ACTION IOFilter_Action:
;
(* Update Functions for pin 1.9 *)

    (* AI filtering for pin X1.09 *)
        AI_u16_DrivetrainTemp_AI := AI_MeanValue(AI_ARR_INDEX,ADR(AI_ARR_u16_DrivetrainTemp_AI),1,50,10);
        AIPU_u16_DrivetrainTemp_AI := AI_MeanValue(AI_ARR_INDEX,ADR(AIPU_ARR_u16_DrivetrainTemp_AI),1,50,10);


(* Update Functions for pin 1.10 *)

    (* AI filtering for pin X1.10 *)
        AI_u16_ChargePlugPresent_AI := AI_MeanValue(AI_ARR_INDEX,ADR(AI_ARR_u16_ChargePlugPresent_AI),1,50,10);
        AIPU_u16_ChargePlugPresent_AI := AI_MeanValue(AI_ARR_INDEX,ADR(AIPU_ARR_u16_ChargePlugPresent_AI),1,50,10);


(* Update Functions for pin 1.11 *)

     (* Debounce filtering to raw DI value of pin 1.11 *)
     G_DebounceDI_q_BatteryInterlockIn_DI(i_In:=DI_RAW_q_BatteryInterlockIn_DI,i_Delay:=30);
     DI_q_BatteryInterlockIn_DI:=G_DebounceDI_q_BatteryInterlockIn_DI.o_Out;

(* Update Functions for pin 1.12 *)

(* Update Functions for pin 1.20 *)

    (* AI filtering for pin X1.20 *)
        AI_u16_Heater1Temperature_AI := AI_MeanValue(AI_ARR_INDEX,ADR(AI_ARR_u16_Heater1Temperature_AI),1,50,10);
        AIPU_u16_Heater1Temperature_AI := AI_MeanValue(AI_ARR_INDEX,ADR(AIPU_ARR_u16_Heater1Temperature_AI),1,50,10);


(* Update Functions for pin 1.21 *)

    (* AI filtering for pin X1.21 *)
        AI_u16_Heater2Temperature_AI := AI_MeanValue(AI_ARR_INDEX,ADR(AI_ARR_u16_Heater2Temperature_AI),1,50,10);
        AIPU_u16_Heater2Temperature_AI := AI_MeanValue(AI_ARR_INDEX,ADR(AIPU_ARR_u16_Heater2Temperature_AI),1,50,10);


(* Update Functions for pin 1.22 *)

(* Update Functions for pin 1.23 *)

(* Update Functions for pin 1.29 *)

(* Update Functions for pin 1.30 *)

(* Update Functions for pin 1.31 *)

(* Update Functions for pin 1.32 *)

(* Update Functions for pin 1.33 *)

(* Update Functions for pin 1.34 *)

(* Update Functions for pin 1.35 *)

(* Update Functions for pin 2.6 *)

     (* Debounce filtering to raw DI value of pin 2.6 *)
     G_DebounceDI_q_Battery1ChargeRq_DI(i_In:=DI_RAW_q_Battery1ChargeRq_DI,i_Delay:=30);
     DI_q_Battery1ChargeRq_DI:=G_DebounceDI_q_Battery1ChargeRq_DI.o_Out;

(* Update Functions for pin 2.7 *)

     (* Debounce filtering to raw DI value of pin 2.7 *)
     G_DebounceDI_q_Battery1DiscahrgeRq_DI(i_In:=DI_RAW_q_Battery1DiscahrgeRq_DI,i_Delay:=30);
     DI_q_Battery1DiscahrgeRq_DI:=G_DebounceDI_q_Battery1DiscahrgeRq_DI.o_Out;

(* Update Functions for pin 2.8 *)

     (* Debounce filtering to raw DI value of pin 2.8 *)
     G_DebounceDI_q_Battery2ChargeRq_DI(i_In:=DI_RAW_q_Battery2ChargeRq_DI,i_Delay:=30);
     DI_q_Battery2ChargeRq_DI:=G_DebounceDI_q_Battery2ChargeRq_DI.o_Out;

(* Update Functions for pin 2.9 *)

     (* Debounce filtering to raw DI value of pin 2.9 *)
     G_DebounceDI_q_Batter2DischargeRq_DI(i_In:=DI_RAW_q_Batter2DischargeRq_DI,i_Delay:=30);
     DI_q_Batter2DischargeRq_DI:=G_DebounceDI_q_Batter2DischargeRq_DI.o_Out;

(* Update Functions for pin 2.13 *)

(* Update Functions for pin 2.14 *)

(* Update Functions for pin 2.15 *)

(* Update Functions for pin 2.17 *)

     (* Debounce filtering to raw DI value of pin 2.17 *)
     G_DebounceDI_q_ChargePlugLockStatus_DI(i_In:=DI_RAW_q_ChargePlugLockStatus_DI,i_Delay:=30);
     DI_q_ChargePlugLockStatus_DI:=G_DebounceDI_q_ChargePlugLockStatus_DI.o_Out;

(* Update Functions for pin 2.17 *)

(* Update Functions for pin 2.18 *)

(* Update Functions for pin 2.19 *)

(* Update Functions for pin 2.20 *)

(* Update Functions for pin 2.23 *)

    (* AI filtering for pin X2.23 *)
        AI_u16_HeaterDiagnose_AI := AI_MeanValue(AI_ARR_INDEX,ADR(AI_ARR_u16_HeaterDiagnose_AI),1,50,10);
        AIPU_u16_HeaterDiagnose_AI := AI_MeanValue(AI_ARR_INDEX,ADR(AIPU_ARR_u16_HeaterDiagnose_AI),1,50,10);


(* Update Functions for pin 2.26 *)

(* Update Functions for pin 2.27 *)

(* Update Functions for pin 2.28 *)

(* Update Functions for pin 2.29 *)

(* Update Functions for pin 2.30 *)

(* Update Functions for pin 2.31 *)

(* Update Functions for pin 2.32 *)

(* Update Functions for pin 2.33 *)

(* Update Functions for pin 2.34 *)

(* Update Functions for pin 2.35 *)

(* Update Functions for pin 3.5 *)

     (* Debounce filtering to raw DI value of pin 3.5 *)
     G_DebounceDI_q_DirectionSwitch_ReverseCrawl_DI(i_In:=DI_RAW_q_DirectionSwitch_ReverseCrawl_DI,i_Delay:=30);
     DI_q_DirectionSwitch_ReverseCrawl_DI:=G_DebounceDI_q_DirectionSwitch_ReverseCrawl_DI.o_Out;

(* Update Functions for pin 3.6 *)

     (* Debounce filtering to raw DI value of pin 3.6 *)
     G_DebounceDI_q_DirectionSwitch_Drive_DI(i_In:=DI_RAW_q_DirectionSwitch_Drive_DI,i_Delay:=30);
     DI_q_DirectionSwitch_Drive_DI:=G_DebounceDI_q_DirectionSwitch_Drive_DI.o_Out;

(* Update Functions for pin 3.7 *)

     (* Debounce filtering to raw DI value of pin 3.7 *)
     G_DebounceDI_q_IlluminiationStatsus_DI(i_In:=DI_RAW_q_IlluminiationStatsus_DI,i_Delay:=30);
     DI_q_IlluminiationStatsus_DI:=G_DebounceDI_q_IlluminiationStatsus_DI.o_Out;

(* Update Functions for pin 3.8 *)

     (* Debounce filtering to raw DI value of pin 3.8 *)
     G_DebounceDI_q_DirectionSwitch_Reverse_DI(i_In:=DI_RAW_q_DirectionSwitch_Reverse_DI,i_Delay:=30);
     DI_q_DirectionSwitch_Reverse_DI:=G_DebounceDI_q_DirectionSwitch_Reverse_DI.o_Out;

(* Update Functions for pin 3.9 *)

     (* Debounce filtering to raw DI value of pin 3.9 *)
     G_DebounceDI_q_DirectionSwitch_DriveCrawl_DI(i_In:=DI_RAW_q_DirectionSwitch_DriveCrawl_DI,i_Delay:=30);
     DI_q_DirectionSwitch_DriveCrawl_DI:=G_DebounceDI_q_DirectionSwitch_DriveCrawl_DI.o_Out;

(* Update Functions for pin 3.10 *)

(* Update Functions for pin 3.11 *)

     (* Debounce filtering to raw DI value of pin 3.11 *)
     G_DebounceDI_q_DirectionSwitch_Neutral_DI(i_In:=DI_RAW_q_DirectionSwitch_Neutral_DI,i_Delay:=30);
     DI_q_DirectionSwitch_Neutral_DI:=G_DebounceDI_q_DirectionSwitch_Neutral_DI.o_Out;

(* Update Functions for pin 3.12 *)

     (* Debounce filtering to raw DI value of pin 3.12 *)
     G_DebounceDI_q_DoorOpen_DI(i_In:=DI_RAW_q_DoorOpen_DI,i_Delay:=30);
     DI_q_DoorOpen_DI:=G_DebounceDI_q_DoorOpen_DI.o_Out;

(* Update Functions for pin 3.14 *)

    (* AI filtering for pin X3.14 *)
        AI_u16_HeaterDiagnose2_AI := AI_MeanValue(AI_ARR_INDEX,ADR(AI_ARR_u16_HeaterDiagnose2_AI),1,50,10);
        AIPU_u16_HeaterDiagnose2_AI := AI_MeanValue(AI_ARR_INDEX,ADR(AIPU_ARR_u16_HeaterDiagnose2_AI),1,50,10);


(* Update Functions for pin 3.15 *)

    (* AI filtering for pin X3.15 *)
        AI_u16_VehicleThrottlePedal1_AI := AI_MeanValue(AI_ARR_INDEX,ADR(AI_ARR_u16_VehicleThrottlePedal1_AI),1,50,10);
        AIPU_u16_VehicleThrottlePedal1_AI := AI_MeanValue(AI_ARR_INDEX,ADR(AIPU_ARR_u16_VehicleThrottlePedal1_AI),1,50,10);



(* Update Functions for pin 3.16 *)

    (* AI filtering for pin X3.16 *)
        AI_u16_VehicleThrottlePedal2_AI := AI_MeanValue(AI_ARR_INDEX,ADR(AI_ARR_u16_VehicleThrottlePedal2_AI),1,50,10);
        AIPU_u16_VehicleThrottlePedal2_AI := AI_MeanValue(AI_ARR_INDEX,ADR(AIPU_ARR_u16_VehicleThrottlePedal2_AI),1,50,10);



(* Update Functions for pin 3.17 *)

(* Update Functions for pin 3.18 *)

(* Update Functions for pin 3.19 *)

(* Update Functions for pin 3.21 *)

(* Update Functions for pin 3.22 *)

     (* Debounce filtering to raw DI value of pin 3.22 *)
     G_DebounceDI_q_VehicleKL15_DI(i_In:=DI_RAW_q_VehicleKL15_DI,i_Delay:=30);
     DI_q_VehicleKL15_DI:=G_DebounceDI_q_VehicleKL15_DI.o_Out;

(* Update Functions for pin 3.23 *)

     (* Debounce filtering to raw DI value of pin 3.23 *)
     G_DebounceDI_q_VehicleKL51_DI(i_In:=DI_RAW_q_VehicleKL51_DI,i_Delay:=30);
     DI_q_VehicleKL51_DI:=G_DebounceDI_q_VehicleKL51_DI.o_Out;

(* Update Functions for pin 3.26 *)

(* Update Functions for pin 3.27 *)

(* Update Functions for pin 3.28 *)

    (* Debounce filtering to raw DI value of pin 3.28 *)
        G_DebounceDI_q_HeaterIn_DI(i_In:=DI_RAW_q_HeaterIn_DI,i_Delay:=30);
        DI_q_HeaterIn_DI:=G_DebounceDI_q_HeaterIn_DI.o_Out;

(* Update Functions for pin 3.29 *)

    (* AI filtering for output voltage measurement in pin X3.29 *)
        AI_q_HeaterOut_DI_Ai := AI_MeanValue(AI_ARR_INDEX,ADR(AI_ARR_q_HeaterOut_DI),1,50,10);


(* Update Functions for pin 3.30 *)

    (* AI filtering for output voltage measurement in pin X3.30 *)
        AI_q_DrivetrainInverterRf1_DO_Ai := AI_MeanValue(AI_ARR_INDEX,ADR(AI_ARR_q_DrivetrainInverterRf1_DO),1,50,10);

(* Update Functions for pin 3.31 *)

    (* AI filtering for output voltage measurement in pin X3.31 *)
        AI_q_DrivetrainInverterRf2_DO_Ai := AI_MeanValue(AI_ARR_INDEX,ADR(AI_ARR_q_DrivetrainInverterRf2_DO),1,50,10);

(* Update Functions for pin 3.32 *)

    (* AI filtering for output voltage measurement in pin X3.32 *)
        AI_q_DrivetrainDCDCInhibit_DO_Ai := AI_MeanValue(AI_ARR_INDEX,ADR(AI_ARR_q_DrivetrainDCDCInhibit_DO),1,50,10);


(* Update Functions for pin 3.33 *)

    (* AI filtering for output voltage measurement in pin X3.33 *)
        AI_q_ChargePlugLED_Green_DO_Ai := AI_MeanValue(AI_ARR_INDEX,ADR(AI_ARR_q_ChargePlugLED_Green_DO),1,50,10);

(* Update Functions for pin 3.34 *)

    (* AI filtering for output voltage measurement in pin X3.34 *)
        AI_q_ChargePlugLED_Blue_DO_Ai := AI_MeanValue(AI_ARR_INDEX,ADR(AI_ARR_q_ChargePlugLED_Blue_DO),1,50,10);

(* Update Functions for pin 3.35 *)

    (* AI filtering for output voltage measurement in pin X3.35 *)
        AI_q_ChargePlugLED_Red_DO_Ai := AI_MeanValue(AI_ARR_INDEX,ADR(AI_ARR_q_ChargePlugLED_Red_DO),1,50,10);
END_ACTION

ACTION IOHandleOutputs_Action:
;

(* AI over current protection for pin X1.09 *)
   IF AI_SET_mA_u16_DrivetrainTemp_AI = TRUE THEN
        (* mA resistor connected set mode correctly *)
        G_AIprotection_X1_09(i_AiInmAMode:= TRUE);
   END_IF
   G_AIprotection_X1_09(
                                                      i_PullUpVoltage := AIPU_RAW_u16_DrivetrainTemp_AI,
                                                      o_ModeSelection =>AI_SET_mA_u16_DrivetrainTemp_AI,
                                                      o_OverCurrentError =>ERR_FLAG_IO_AI_OVER_CURRENT_X1_09);

(* AI over current protection for pin X1.10 *)
   IF AI_SET_mA_u16_ChargePlugPresent_AI = TRUE THEN
        (* mA resistor connected set mode correctly *)
        G_AIprotection_X1_10(i_AiInmAMode:= TRUE);
   END_IF
   G_AIprotection_X1_10(
                                                      i_PullUpVoltage := AIPU_RAW_u16_ChargePlugPresent_AI,
                                                      o_ModeSelection =>AI_SET_mA_u16_ChargePlugPresent_AI,
                                                      o_OverCurrentError =>ERR_FLAG_IO_AI_OVER_CURRENT_X1_10);

(* AI over current protection for pin X1.20 *)
   IF AI_SET_mA_u16_Heater1Temperature_AI = TRUE THEN
        (* mA resistor connected set mode correctly *)
        G_AIprotection_X1_20(i_AiInmAMode:= TRUE);
   END_IF
   G_AIprotection_X1_20(
                                                      i_PullUpVoltage := AIPU_RAW_u16_Heater1Temperature_AI,
                                                      o_ModeSelection =>AI_SET_mA_u16_Heater1Temperature_AI,
                                                      o_OverCurrentError =>ERR_FLAG_IO_AI_OVER_CURRENT_X1_20);

(* AI over current protection for pin X1.20 *)
   IF AI_SET_mA_u16_Heater2Temperature_AI = TRUE THEN
        (* mA resistor connected set mode correctly *)
        G_AIprotection_X1_21(i_AiInmAMode:= TRUE);
   END_IF
   G_AIprotection_X1_21(
                                                      i_PullUpVoltage := AIPU_RAW_u16_Heater2Temperature_AI,
                                                      o_ModeSelection =>AI_SET_mA_u16_Heater2Temperature_AI,
                                                      o_OverCurrentError =>ERR_FLAG_IO_AI_OVER_CURRENT_X1_21);

(* AI over current protection for pin X2.23 *)
   IF AI_SET_mA_u16_HeaterDiagnose_AI = TRUE THEN
        (* mA resistor connected set mode correctly *)
        G_AIprotection_X2_23(i_AiInmAMode:= TRUE);
   END_IF
   G_AIprotection_X2_23(
                                                      i_PullUpVoltage := AIPU_RAW_u16_HeaterDiagnose_AI,
                                                      o_ModeSelection =>AI_SET_mA_u16_HeaterDiagnose_AI,
                                                      o_OverCurrentError =>ERR_FLAG_IO_AI_OVER_CURRENT_X2_23);

(* AI over current protection for pin X3.14 *)
   IF AI_SET_mA_u16_HeaterDiagnose2_AI = TRUE THEN
        (* mA resistor connected set mode correctly *)
        G_AIprotection_X3_14(i_AiInmAMode:= TRUE);
   END_IF
   G_AIprotection_X3_14(
                                                      i_PullUpVoltage := AIPU_RAW_u16_HeaterDiagnose2_AI,
                                                      o_ModeSelection =>AI_SET_mA_u16_HeaterDiagnose2_AI,
                                                      o_OverCurrentError =>ERR_FLAG_IO_AI_OVER_CURRENT_X3_14);

(* AI over current protection for pin X3.15 *)
   IF AI_SET_mA_u16_VehicleThrottlePedal1_AI = TRUE THEN
        (* mA resistor connected set mode correctly *)
        G_AIprotection_X3_15(i_AiInmAMode:= TRUE);
   END_IF
   G_AIprotection_X3_15(
                                                      i_PullUpVoltage := AIPU_RAW_u16_VehicleThrottlePedal1_AI,
                                                      o_ModeSelection =>AI_SET_mA_u16_VehicleThrottlePedal1_AI,
                                                      o_OverCurrentError =>ERR_FLAG_IO_AI_OVER_CURRENT_X3_15);

(* AI over current protection for pin X3.16 *)
   IF AI_SET_mA_u16_VehicleThrottlePedal2_AI = TRUE THEN
        (* mA resistor connected set mode correctly *)
        G_AIprotection_X3_16(i_AiInmAMode:= TRUE);
   END_IF
   G_AIprotection_X3_16(
                                                      i_PullUpVoltage := AIPU_RAW_u16_VehicleThrottlePedal2_AI,
                                                      o_ModeSelection =>AI_SET_mA_u16_VehicleThrottlePedal2_AI,
                                                      o_OverCurrentError =>ERR_FLAG_IO_AI_OVER_CURRENT_X3_16);
END_ACTION

ACTION Main_Application_Action:
(* Call user application *)
Main();
END_ACTION

ACTION Other_Action:
// Target specific. Not available.
END_ACTION

ACTION Other_EpecOut_Action:
(* tag EPEC_OUT_OTHER *)

(* If reset flag set --> restart unit *)
IF G_RESET_MODULE THEN
    EPEC_5000EXT.BOOT_APPLICATION_KILL_RTS();
END_IF

(* Block actions if voltage level is under defined limit *)
IF G_HWDiagnostics.o_SupplyVoltage1 > G_LowLimitForParameterSaving THEN

	
    IF G_CounterRestoreCmdOld<> G_SaveOD_RestoreCommsCounter THEN 
         (* Restore command given trough CANopen *)
         G_CounterRestoreCmdOld := G_SaveOD_RestoreCommsCounter;   
         SystemParameters.RestoreDefaultData();
         G_SystemInfo.EthernetConfiguration := SystemParameters.i_Ethernet;  
         G_SystemInfo.CAN1_Comms := SystemParameters.i_CAN1;
         G_SystemInfo.CAN2_Comms := SystemParameters.i_CAN2;      
         G_SystemInfo.CAN3_Comms := SystemParameters.i_CAN3;      
         G_SystemInfo.CAN4_Comms := SystemParameters.i_CAN4;      
    END_IF
    
    IF G_CounterSaveCmdOld  <> G_SaveOD_SaveCommsCounter THEN
        (* Save command given trough CANopen *)
        G_CounterSaveCmdOld  := G_SaveOD_SaveCommsCounter;
        SystemParameters.i_Ethernet := G_SystemInfo.EthernetConfiguration;
        SystemParameters.i_CAN1 := G_SystemInfo.CAN1_Comms;
        SystemParameters.i_CAN2 := G_SystemInfo.CAN2_Comms;
        SystemParameters.i_CAN3 := G_SystemInfo.CAN3_Comms;
        SystemParameters.i_CAN4 := G_SystemInfo.CAN4_Comms;
        SystemParameters.WriteData();
    END_IF
END_IF
END_ACTION

END_PROGRAM

// Application/UserCode/Functions/Update
(*==============================================================================================================*)
(*     Function to handle state updates                                                                         *)
(*==============================================================================================================*)
FUNCTION Update : BOOL
VAR_INPUT
 ptUp        : POINTER TO tUpdate; // Pointer to screen update

END_VAR
VAR
END_VAR

(*==============================================================================================================*)
(*     Function to handle state updates                                                                         *)
(*==============================================================================================================*)
IF (ptUp^.Next <> ptUp^.Step) THEN                         // New State Requested?	
	ptUp^.Last			:= ptUp^.Step;                     // Save Current State
	ptUp^.Step			:= ptUp^.Next;                     // Set New State
	ptUp^.Seq  			:= (ptUp^.Seq * 256) + ptUp^.Next; // Shift In New State
	ptUp^.Tmr			:= 0;                              // Reset State Timer
ELSIF (ptUp^.Tmr <> 65535) THEN                            // Timer Less than max?
	ptUp^.Tmr			:= (ptUp^.Tmr + 1);                // Increment Timer
END_IF

END_FUNCTION

// Application/UserCode/Main Program/MainInit
PROGRAM MainInit
VAR_OUTPUT
	o_MainInitReady: BOOL := FALSE;
END_VAR


(*Check if CAN bitrate in device communication parameters is 500kbit/s.
If not, set it to 500 kbit/s *)
EPEC_5050INT.SystemParameters.ReadData();
IF EPEC_5050INT.SystemParameters.i_CAN1[3] <> gu16_CAN1_BaudRate THEN
                             EPEC_5050INT.SystemParameters.i_CAN1[3] := gu16_CAN1_BaudRate;
                             EPEC_5050INT.SystemParameters.WriteData();
END_IF
IF EPEC_5050INT.SystemParameters.i_CAN2[3] <> gu16_CAN2_BaudRate THEN
                             EPEC_5050INT.SystemParameters.i_CAN2[3] := gu16_CAN2_BaudRate;
                             EPEC_5050INT.SystemParameters.WriteData();
END_IF
IF EPEC_5050INT.SystemParameters.i_CAN3[3] <> gu16_CAN3_BaudRate THEN
                             EPEC_5050INT.SystemParameters.i_CAN3[3] := gu16_CAN3_BaudRate;
                             EPEC_5050INT.SystemParameters.WriteData();
END_IF
IF EPEC_5050INT.SystemParameters.i_CAN4[3] <> gu16_CAN4_BaudRate THEN
                             EPEC_5050INT.SystemParameters.i_CAN4[3] := gu16_CAN4_BaudRate;
                             EPEC_5050INT.SystemParameters.WriteData();
END_IF

o_MainInitReady := TRUE;

END_PROGRAM

// Application/UserCode/Main Program/Main
PROGRAM Main
VAR
	hq_ManualChangeBaud	:	BOOL;
	hton_Timer	:	TON;
END_VAR

/// User code should be added to POU named as Main.
(*Reallocation of Outputs to correct variables*)
IO_Reconfiguration();


(*Check to make sure that the component selection hasn't been changed*)
ComponentSelection();

(*******************************************************)
(*Receive Routines*)
Sevcon_Steer_Rx();
Sevcon2_Rx();
Brusa1_Rx();
Brusa2_Rx();
MCU_Rx();
OrionBMS1_Rx();
OrionBMS2_Rx();
BELDCDC_Rx();
BELDCDC_Tx();
BELDCDC_TxConversion();
HMI_Rx();
CAN1_Rx();
CAN3_Rx();
CAN4_Rx();
ePTO_Rx();
Chassis_Parameters();
Cooling_Fan();
(*******************************************************)
(*Control*)
FaultDetection();
System_StateSpace();
ContactorControl();
GearSelection();
Dennis_Regen();
(*Battery Selection*)
IF (gu8_BMSType = BMS_ORION) THEN
	Orion_Control();
END_IF
BMSData();
MCU_Control();
BELDCDC_Control();
Brusa();
Sevcon_Steer_Control();
Sevcon2_Control();
Heater_Control();
ePTO_Control();
Project_Infomation();
(*******************************************************)

(*Transmit Routines*)
IF (gu8_BMSType = BMS_ORION) THEN
	OrionBMS_Tx();

END_IF
Sevcon_Steer_Tx();
Sevcon2_Tx();
MCU_Tx();
Brusa1_Tx();
Brusa2_Tx();
CAN4_Tx();
CAN1_Tx();
Heater_Tx();
Heater_Rx();
EPTO_Tx();
CAN3_Tx();

(*******************************************************)

(*Chassis specific transmit/persistent messages*)
IF gu8_ChassisType = CHASSIS_DENNIS THEN
	KB_Tx();
	gq_APU_Installed	:=	FALSE;
	gq_Daimler_PowerShift_Installed	:=	FALSE;
	gq_Allison_Pad_Override	:=	TRUE;
END_IF

IF gu8_ChassisType = CHASSIS_ESTARGLIDER THEN
	CAN1_TCMs_Tx();
	
	gq_APU_Installed	:=	TRUE;
END_IF

IF gu8_ChassisType = CHASSIS_IVECO THEN
	gq_APU_Installed	:=	FALSE;
	gq_Daimler_PowerShift_Installed	:=	FALSE;
	gq_Allison_Pad_Override	:=	FALSE;
END_IF

METHOD IO_Reconfiguration
VAR_INPUT
END_VAR
IF E_Stop_Installed = TRUE THEN
gq_EStop	:= (NOT DI_q_DirectionSwitch_ReverseCrawl_DI OR HMI_Rx.gq_HMI_EStop_Bad); (*OR changed to AND Latch the Estop on unless you go out of drive*)
END_IF

gq_BMS1_AuxPosContactor		:=	DI_q_Battery1ChargeRq_DI; (*Batt1 +ve contactor status feedback for DO_q_BatteryDischargeMain_DO*)
gq_BMS1_AuxNegContactor		:=	DI_q_Battery1DiscahrgeRq_DI; (*Batt1 -ve contactor status (BMS Controlled Contactor)*)
gq_BMS2_AuxPosContactor		:=	DI_q_Battery2ChargeRq_DI; (*Batt2 +ve contactor Status (BMS Controlled Contactor)*)
gq_BMS2_AuxNegContactor		:=	DI_q_Batter2DischargeRq_DI; (*Batt2 -ve contactor Status (BMS Controlled Contactor)*)

IF (gq_BodyStepInstalled = TRUE) THEN
	gq_BodySteps	:=	NOT(DOS_q_DrievtrainAirCompressor_DO);
END_IF

(*Using heater control for the reverse lights*)
PWFM_FREQ_u32_HeaterControl_PWFM := 3000;
IF (gq_ReverseLights = TRUE) THEN
	PWFM_RATIO_u32_HeaterControl_PWFM	:=	1000;
ELSE
	PWFM_RATIO_u32_HeaterControl_PWFM	:=	0;
END_IF

DO_q_AirPressureReliefValve_DO	:=	gq_ePTO_FanEnable;
END_METHOD

END_PROGRAM

// Application/UserCode/Main Program/ComponentSelection
PROGRAM ComponentSelection
VAR
	ChangeComponentSelection_Rx	:	Receive_CAN4_EXD;
	hu8_MultiplexSelector		:	USINT;
END_VAR
VAR CONSTANT
	CHASSIS_SELECT				:	USINT	:=	1;
	CHARGER_SELECT				:	USINT	:=	2;
	BMS_SELECT					:	USINT	:=	4;
	CAN1_BAUDRATE				:	USINT	:=	8;
	CAN2_BAUDRATE				:	USINT	:=	16;
	CAN3_BAUDRATE				:	USINT	:=	32;
	CAN4_BAUDRATE				:	USINT	:=	64;
	REARSTEER_INST				:	USINT	:=	18;
	SPEED_CAL					:	USINT	:=	69;
	TIREPROFILE					:	USINT	:=	70;
	
	SELECTBAUD250K				:	USINT	:=	1;
	SELECTBAUD500K				:	USINT	:=	2;
	BAUD250K					:	UINT	:=	250;
	BAUD500K					:	UINT	:=	500;
	
	
END_VAR


ChangeComponentSelection_Rx(u32_COBID	:=	16#18FFFF01,
											q_NewData => ,
											au8_Data => ,
											u8_Length => 			);
				
				
hu8_MultiplexSelector	:=	ChangeComponentSelection_Rx.au8_Data[0];				
				
CASE hu8_MultiplexSelector OF
	CHASSIS_SELECT:
		gu8_ChassisType	:=	ChangeComponentSelection_Rx.au8_Data[1];	
	CHARGER_SELECT:
		gu8_ChargerType	:=	ChangeComponentSelection_Rx.au8_Data[2];
	BMS_SELECT:
		gu8_BMSType		:=	ChangeComponentSelection_Rx.au8_Data[3];
	CAN1_BAUDRATE:
		IF (ChangeComponentSelection_Rx.au8_Data[4] = SELECTBAUD250K) THEN
			gu16_CAN1_BaudRate	:=	BAUD250K;
		ELSIF (ChangeComponentSelection_Rx.au8_Data[4] = SELECTBAUD500K) THEN
			gu16_CAN1_BaudRate	:=	BAUD500K;
		END_IF
	CAN2_BAUDRATE:
		IF (ChangeComponentSelection_Rx.au8_Data[4] = SELECTBAUD250K) THEN
			gu16_CAN2_BaudRate	:=	BAUD250K;
		ELSIF (ChangeComponentSelection_Rx.au8_Data[4] = SELECTBAUD500K) THEN
			gu16_CAN2_BaudRate	:=	BAUD500K;
		END_IF
	CAN3_BAUDRATE:
		IF (ChangeComponentSelection_Rx.au8_Data[4] = SELECTBAUD250K) OR (gu8_ChassisType = CHASSIS_DENNIS OR gu8_ChassisType = CHASSIS_IVECO) THEN
			gu16_CAN3_BaudRate	:=	BAUD250K;
		ELSIF (ChangeComponentSelection_Rx.au8_Data[4] = SELECTBAUD500K) OR (gu8_ChassisType = CHASSIS_ESTARGLIDER) THEN
			gu16_CAN3_BaudRate	:=	BAUD500K;
		END_IF
	CAN4_BAUDRATE:
		IF (ChangeComponentSelection_Rx.au8_Data[4] = SELECTBAUD250K) THEN
			gu16_CAN4_BaudRate	:=	BAUD250K;
		ELSIF (ChangeComponentSelection_Rx.au8_Data[4] = SELECTBAUD500K) THEN
			gu16_CAN4_BaudRate	:=	BAUD500K;
		END_IF
	(*REARSTEER_INST:
		gq_RearSteer_Installed	:=	ChangeComponentSelection_Rx.au8_Data[5].0;*)
	SPEED_CAL:
		IF (ChangeComponentSelection_Rx.au8_Data[1] <> 0 OR ChangeComponentSelection_Rx.au8_Data[2] <> 0) THEN
			gu16_GearRatio_PreCF		:=	USINT_TO_UINT(ChangeComponentSelection_Rx.au8_Data[1]) + SHL(USINT_TO_UINT(ChangeComponentSelection_Rx.au8_Data[2]), 8);
		END_IF
		IF (ChangeComponentSelection_Rx.au8_Data[3] <> 0 OR ChangeComponentSelection_Rx.au8_Data[4] <> 0) THEN
			gu16_DyfRatio_PreCF			:=	USINT_TO_UINT(ChangeComponentSelection_Rx.au8_Data[3]) + SHL(USINT_TO_UINT(ChangeComponentSelection_Rx.au8_Data[4]), 8);
		END_IF
	TIREPROFILE:
		gu16_TireWidth_mm			:=	USINT_TO_UINT(ChangeComponentSelection_Rx.au8_Data[1]) + SHL(USINT_TO_UINT(ChangeComponentSelection_Rx.au8_Data[2]), 8);
		gu8_TireProfile_Perc		:=	ChangeComponentSelection_Rx.au8_Data[3];
		gu16_WheelDiameter_PreCF	:=	USINT_TO_UINT(ChangeComponentSelection_Rx.au8_Data[4]) + SHL(USINT_TO_UINT(ChangeComponentSelection_Rx.au8_Data[5]), 8);
ELSE
	;
END_CASE

END_PROGRAM

// Application/UserCode/CAN Function Blocks/CAN4/Receive_CAN4_EXD
FUNCTION_BLOCK Receive_CAN4_EXD
VAR_INPUT
	u32_COBID	:	DWORD;
END_VAR
VAR_OUTPUT
	q_NewData	:	BOOL;
	au8_Data	:	ARRAY [0..7] OF BYTE;
	u8_Length	:	BYTE;
END_VAR
VAR
	hq_Initialise	:	BOOL	:=	FALSE;
	ht_RxMessage	:	t_CANReceive;
	ht_MsgRx		:	Callback_Receive_CAN1;
END_VAR



IF (hq_Initialise = FALSE) THEN
	(*
	IF (u32_COBID > 16#7FF) THEN
		(*29 bit*)
		;
	ELSE
		(*11 bit*)
		;
	END_IF
	*)
	(*
	(*11 bit*)
	G_CAN4_Channel.AddCOBID(i_CobId := u32_COBID,
							i_itfCallback := ht_RxMessage,
							i_Argument := ADR(ht_RxMessage));
	*)
	(*29 bit*)
	G_CAN4_Channel.AddCOBID(i_CobId := u32_COBID OR EPEC_CANVXD.MASK_29BIT,
							i_itfCallback := ht_MsgRx,
							i_Argument := ADR(ht_RxMessage));
	G_CAN4_Channel.SetMask(i_CobID := u32_COBID OR EPEC_CANVXD.MASK_29BIT, i_Mask := 16#18FEF1F2 OR EPEC_CANVXD.MASK_29BIT);

	hq_Initialise	:=	TRUE;
END_IF


IF (ht_RxMessage.q_NewDataRxed = TRUE) THEN
	au8_Data	:=	ht_RxMessage.Data;
	u8_Length	:=	ht_RxMessage.Len;
	q_NewData	:=	TRUE;
	ht_RxMessage.q_NewDataRxed	:=	FALSE;
ELSE
	q_NewData	:=	FALSE;
END_IF

END_FUNCTION_BLOCK

// Application/UserCode/CAN Function Blocks/CAN1/Callback_Receive_CAN1
FUNCTION_BLOCK Callback_Receive_CAN1 IMPLEMENTS
EPEC_CANVXD.IReceiveCallback
VAR_INPUT	
END_VAR
VAR_OUTPUT
END_VAR
VAR
END_VAR

METHOD Receive
VAR_INPUT
	(* Pointer to the CAN message *)
	i_pMsg	: POINTER TO EPEC_CANVXD.Msg;
	(* User specific argument. This is set in AddCOBID i_Argument. *)
	i_Argument	: DWORD;
END_VAR
VAR
	t_pRxMessage : POINTER TO t_CANReceive;
END_VAR


t_pRxMessage				:=	i_Argument;
t_pRxMessage^.q_NewDataRxed	:=	TRUE;
t_pRxMessage^.Data			:=	i_pMsg^.Data;
t_pRxMessage^.ID			:=	i_pMsg^.ID;
t_pRxMessage^.Len			:=	i_pMsg^.Len;
END_METHOD

END_FUNCTION_BLOCK

// Application/UserCode/Sevcon_PSP/Sevcon_Steer_Rx
PROGRAM Sevcon_Steer_Rx
VAR
	TorqueStatus1_Rx	:	Receive_CAN2_EXD;
	TorqueStatus2_Rx	:	Receive_CAN2_EXD;
	TempStatus_Rx		:	Receive_CAN2_EXD;
	FaultStatus_Rx		:	Receive_CAN2_EXD;
	EncoderStatus_Rx	:	Receive_CAN2_EXD;
	DeubgCurrents_Rx	:	Receive_CAN2_EXD;
	DebugTemps1_Rx		:	Receive_CAN2_EXD;
	DebugTemps2_Rx		:	Receive_CAN2_EXD;
	DebugPMACControl_Rx	:	Receive_CAN2_EXD;
	DebugFVControl_Rx	:	Receive_CAN2_EXD;
	
	TorqueStatus1_Rx_Timer		:	TON;
	TorqueStatus2_Rx_Timer		:	TON;
	TempStatus_Rx_Timer			:	TON;
	FaultStatus_Rx_Timer		:	TON;
	EncoderStatus_Rx_Timer		:	TON;
	DeubgCurrents_Rx_Timer		:	TON;
	DebugTemps1_Rx_Timer		:	TON;
	DebugTemps2_Rx_Timer		:	TON;
	DebugPMACControl_Rx_Timer	:	TON;
	DebugFVControl_Rx_Timer		:	TON;
END_VAR


TorqueStatus1_Rx(u32_COBID	:=	16#1918FF71,
				q_NewData => ,
				au8_Data => ,
				u8_Length => 			);

TorqueStatus2_Rx(u32_COBID	:=	16#1919FF71,
				q_NewData => ,
				au8_Data => ,
				u8_Length => 			);

TempStatus_Rx(u32_COBID	:=	16#191AFF71,
				q_NewData => ,
				au8_Data => ,
				u8_Length => 			);

FaultStatus_Rx(u32_COBID	:=	16#191BFF71,
				q_NewData => ,
				au8_Data => ,
				u8_Length => 			);

EncoderStatus_Rx(u32_COBID	:=	16#191CFF71,
				q_NewData => ,
				au8_Data => ,
				u8_Length => 			);

DeubgCurrents_Rx(u32_COBID	:=	16#1928FF71,
				q_NewData => ,
				au8_Data => ,
				u8_Length => 			);

DebugTemps1_Rx(u32_COBID	:=	16#192AFF71,
				q_NewData => ,
				au8_Data => ,
				u8_Length => 			);

DebugTemps2_Rx(u32_COBID	:=	16#192BFF71,
				q_NewData => ,
				au8_Data => ,
				u8_Length => 			);

DebugPMACControl_Rx(u32_COBID	:=	16#192CFF71,
				q_NewData => ,
				au8_Data => ,
				u8_Length => 			);

DebugFVControl_Rx(u32_COBID	:=	16#192DFF71,
				q_NewData => ,
				au8_Data => ,
				u8_Length => 			);				

			
				
gs16_Sevcon1_TorqueMeasured_Rx			:=	USINT_TO_INT(TorqueStatus1_Rx.au8_Data[0]) +
											SHL(USINT_TO_INT(TorqueStatus1_Rx.au8_Data[1]), 8);
gs16_Sevcon1_SpeedMeasured				:=	USINT_TO_INT(TorqueStatus1_Rx.au8_Data[2]) +
											SHL(USINT_TO_INT(TorqueStatus1_Rx.au8_Data[3]), 8);
gs16_Sevcon1_DCLink_Current				:=	USINT_TO_INT(TorqueStatus1_Rx.au8_Data[4]) +
											SHL(USINT_TO_INT(TorqueStatus1_Rx.au8_Data[5]), 8);
gu8_Sevcon1_SEQ_Torque					:=	TorqueStatus1_Rx.au8_Data[6];
gu8_Sevcon1_CS_Torque					:=	TorqueStatus1_Rx.au8_Data[7];

gs16_Sevcon1_TorqueAvailableForward_Rx	:=	USINT_TO_INT(TorqueStatus2_Rx.au8_Data[0]) +
											SHL(USINT_TO_INT(TorqueStatus2_Rx.au8_Data[1]), 8);
gs16_Sevcon1_TorqueAvailableReverse_Rx	:=	USINT_TO_INT(TorqueStatus2_Rx.au8_Data[2]) +
											SHL(USINT_TO_INT(TorqueStatus2_Rx.au8_Data[3]), 8);
gu8_Sevcon1_InverterStatus				:=	TorqueStatus2_Rx.au8_Data[4];
gu8_Sevcon1_TorqueLimitCode				:=	TorqueStatus2_Rx.au8_Data[5];
gu8_Sevcon1_SEQ_Status					:=	TorqueStatus2_Rx.au8_Data[6];
gu8_Sevcon1_CS_Status					:=	TorqueStatus2_Rx.au8_Data[7];

gs16_Sevcon1_TempRemaining				:=	USINT_TO_INT(TempStatus_Rx.au8_Data[0]) +
											SHL(USINT_TO_INT(TempStatus_Rx.au8_Data[1]), 8);
gs16_Sevcon1_MotorTemp					:=	USINT_TO_INT(TempStatus_Rx.au8_Data[2]) +
											SHL(USINT_TO_INT(TempStatus_Rx.au8_Data[3]), 8);
gs16_Sevcon1_DCLink_Voltage_Rx			:=	USINT_TO_INT(TempStatus_Rx.au8_Data[4]) +
											SHL(USINT_TO_INT(TempStatus_Rx.au8_Data[5]), 8);
gu8_Sevcon1_SEQ_Temp					:=	TempStatus_Rx.au8_Data[6];
gu8_Sevcon1_CS_Temp						:=	TempStatus_Rx.au8_Data[7];

gs16_Sevcon1_FaultCode					:=	USINT_TO_INT(FaultStatus_Rx.au8_Data[0]) +
											SHL(USINT_TO_INT(FaultStatus_Rx.au8_Data[1]), 8);
gs32_Sevcon1_FaultData					:=	USINT_TO_DINT(FaultStatus_Rx.au8_Data[2]) +
											SHL(USINT_TO_DINT(FaultStatus_Rx.au8_Data[3]), 8) +
											SHL(USINT_TO_DINT(FaultStatus_Rx.au8_Data[4]), 16) +
											SHL(USINT_TO_DINT(FaultStatus_Rx.au8_Data[5]), 24);
gu8_Sevcon1_SEQ_Fault					:=	FaultStatus_Rx.au8_Data[6];
gu8_Sevcon1_CS_Fault					:=	FaultStatus_Rx.au8_Data[7];

gs32_Sevcon1_EncoderPosition_Rx			:=	USINT_TO_DINT(EncoderStatus_Rx.au8_Data[0]) +
											SHL(USINT_TO_DINT(EncoderStatus_Rx.au8_Data[1]), 8) +
											SHL(USINT_TO_DINT(EncoderStatus_Rx.au8_Data[2]), 16) +
											SHL(USINT_TO_DINT(EncoderStatus_Rx.au8_Data[3]), 24);

gs16_Sevcon1_Debug_Id_Act_Rx			:=	USINT_TO_INT(DeubgCurrents_Rx.au8_Data[0]) +
											SHL(USINT_TO_INT(DeubgCurrents_Rx.au8_Data[1]), 8);
gs16_Sevcon1_Debug_Iq_Act_Rx			:=	USINT_TO_INT(DeubgCurrents_Rx.au8_Data[2]) +
											SHL(USINT_TO_INT(DeubgCurrents_Rx.au8_Data[3]), 8);
gs16_Sevcon1_Debug_Id_Ref_Rx			:=	USINT_TO_INT(DeubgCurrents_Rx.au8_Data[4]) +
											SHL(USINT_TO_INT(DeubgCurrents_Rx.au8_Data[5]), 8);
gs16_Sevcon1_Debug_Iq_Ref_Rx			:=	USINT_TO_INT(DeubgCurrents_Rx.au8_Data[6]) +
											SHL(USINT_TO_INT(DeubgCurrents_Rx.au8_Data[7]), 8);

gu8_Sevcon1_Debug_Temp_Junction0		:=	DebugTemps1_Rx.au8_Data[0];
gu8_Sevcon1_Debug_Temp_Junction1		:=	DebugTemps1_Rx.au8_Data[1];
gu8_Sevcon1_Debug_Temp_Junction2		:=	DebugTemps1_Rx.au8_Data[2];
gu8_Sevcon1_Debug_Temp_Junction3		:=	DebugTemps1_Rx.au8_Data[3];
gu8_Sevcon1_Debug_Temp_Junction4		:=	DebugTemps1_Rx.au8_Data[4];
gu8_Sevcon1_Debug_Temp_Junction5		:=	DebugTemps1_Rx.au8_Data[5];
gu8_Sevcon1_Debug_Temp_MotorMeasured	:=	DebugTemps1_Rx.au8_Data[6];
gu8_Sevcon1_Debug_Temp_MotorEstimate	:=	DebugTemps1_Rx.au8_Data[7];

gu8_Sevcon1_Debug_Temp_CapEstimateFast	:=	DebugTemps2_Rx.au8_Data[0];
gu8_Sevcon1_Debug_Temp_Track			:=	DebugTemps2_Rx.au8_Data[1];
gu8_Sevcon1_Debug_Temp_CapEstimateSlow	:=	DebugTemps2_Rx.au8_Data[2];
gu8_Sevcon1_Debug_Temp_Heatsink			:=	DebugTemps2_Rx.au8_Data[3];
gu8_Sevcon1_Debug_Temp_DeltaTj			:=	DebugTemps2_Rx.au8_Data[4];
gu8_Sevcon1_Debug_Temp_Normalised		:=	DebugTemps2_Rx.au8_Data[5];
gu8_Sevcon1_Debug_Temp_Coolant			:=	DebugTemps2_Rx.au8_Data[6];
gu8_Sevcon1_Debug_Temp_Winding			:=	DebugTemps2_Rx.au8_Data[7];

gs16_Sevcon1_Debug_MaxFlux				:=	USINT_TO_INT(DebugPMACControl_Rx.au8_Data[0]) +
											SHL(USINT_TO_INT(DebugPMACControl_Rx.au8_Data[1]), 8);
gs16_Sevcon1_Debug_IvLim				:=	USINT_TO_INT(DebugPMACControl_Rx.au8_Data[2]) +
											SHL(USINT_TO_INT(DebugPMACControl_Rx.au8_Data[3]), 8);
gs16_Sevcon1_Debug_IqMax				:=	USINT_TO_INT(DebugPMACControl_Rx.au8_Data[4]) +
											SHL(USINT_TO_INT(DebugPMACControl_Rx.au8_Data[5]), 8);
gs16_Sevcon1_Debug_Ls_Rx				:=	USINT_TO_INT(DebugPMACControl_Rx.au8_Data[6]) +
											SHL(USINT_TO_INT(DebugPMACControl_Rx.au8_Data[7]), 8);

gs16_Sevcon1_Debug_Slip_Rx				:=	USINT_TO_INT(DebugFVControl_Rx.au8_Data[0]) +
											SHL(USINT_TO_INT(DebugFVControl_Rx.au8_Data[1]), 8);
gs16_Sevcon1_Debug_LmSat_Rx				:=	USINT_TO_INT(DebugFVControl_Rx.au8_Data[2]) +
											SHL(USINT_TO_INT(DebugFVControl_Rx.au8_Data[3]), 8);
gs16_Sevcon1_Debug_IqMax2				:=	USINT_TO_INT(DebugFVControl_Rx.au8_Data[4]) +
											SHL(USINT_TO_INT(DebugFVControl_Rx.au8_Data[5]), 8);
gs16_Sevcon1_Debug_RecipFlux			:=	USINT_TO_INT(DebugFVControl_Rx.au8_Data[6]) +
											SHL(USINT_TO_INT(DebugFVControl_Rx.au8_Data[7]), 8);


TorqueStatus1_Rx_Timer(IN := NOT(TorqueStatus1_Rx.q_NewData), PT := T#3S);
TorqueStatus2_Rx_Timer(IN := NOT(TorqueStatus2_Rx.q_NewData), PT := T#3S);
TempStatus_Rx_Timer(IN := NOT(TempStatus_Rx.q_NewData), PT := T#3S);
FaultStatus_Rx_Timer(IN := NOT(FaultStatus_Rx.q_NewData), PT := T#3S);
EncoderStatus_Rx_Timer(IN := NOT(EncoderStatus_Rx.q_NewData), PT := T#3S);
DeubgCurrents_Rx_Timer(IN := NOT(DeubgCurrents_Rx.q_NewData), PT := T#3S);
DebugTemps1_Rx_Timer(IN := NOT(DebugTemps1_Rx.q_NewData), PT := T#3S);
DebugTemps2_Rx_Timer(IN := NOT(DebugTemps2_Rx.q_NewData), PT := T#3S);
DebugPMACControl_Rx_Timer(IN := NOT(DebugPMACControl_Rx.q_NewData), PT := T#3S);
DebugFVControl_Rx_Timer(IN := NOT(DebugFVControl_Rx.q_NewData), PT := T#3S);
IF (TorqueStatus1_Rx_Timer.Q = TRUE AND TorqueStatus2_Rx_Timer.Q = TRUE AND TempStatus_Rx_Timer.Q = TRUE AND
	FaultStatus_Rx_Timer.Q = TRUE AND EncoderStatus_Rx_Timer.Q = TRUE AND DeubgCurrents_Rx_Timer.Q = TRUE AND
	DebugTemps1_Rx_Timer.Q = TRUE AND DebugTemps2_Rx_Timer.Q = TRUE AND DebugPMACControl_Rx_Timer.Q = TRUE AND
	DebugFVControl_Rx_Timer.Q = TRUE) THEN
	gq_Sevcon1_CommsLoss	:=	TRUE;
ELSE
	gq_Sevcon1_CommsLoss	:=	FALSE;
END_IF
										
Sevcon_Steer_RxConversion();

END_PROGRAM

// Application/UserCode/Sevcon_PSP/Sevcon_Steer_RxConversion
PROGRAM Sevcon_Steer_RxConversion
VAR
END_VAR
VAR CONSTANT
	SIXTEENTH_CF	:	REAL	:=	0.0625;
END_VAR




gr_Sevcon1_TorqueMeasured			:=	gs16_Sevcon1_TorqueMeasured_Rx * SIXTEENTH_CF;
gr_Sevcon1_TorqueAvailableForward	:=	gs16_Sevcon1_TorqueAvailableForward_Rx * SIXTEENTH_CF;
gr_Sevcon1_TorqueAvailableReverse	:=	gs16_Sevcon1_TorqueAvailableReverse_Rx * SIXTEENTH_CF;
gr_Sevcon1_DCLink_Voltage			:=	gs16_Sevcon1_DCLink_Voltage_Rx * SIXTEENTH_CF;
gr_Sevcon1_EncoderPosition			:=	LREAL_TO_REAL(gs32_Sevcon1_EncoderPosition_Rx * (1.5287890625 * EXPT(10, -5)));
gr_Sevcon1_Debug_Id_Act				:=	gs16_Sevcon1_Debug_Id_Act_Rx * SIXTEENTH_CF;
gr_Sevcon1_Debug_Iq_Act				:=	gs16_Sevcon1_Debug_Iq_Act_Rx * SIXTEENTH_CF;
gr_Sevcon1_Debug_Id_Ref				:=	gs16_Sevcon1_Debug_Id_Ref_Rx * SIXTEENTH_CF;
gr_Sevcon1_Debug_Iq_Ref				:=	gs16_Sevcon1_Debug_Iq_Ref_Rx * SIXTEENTH_CF;
gr_Sevcon1_Debug_Ls					:=	LREAL_TO_REAL(gs16_Sevcon1_Debug_Ls_Rx * (5.960464477539 * EXPT(10, -8)));
gr_Sevcon1_Debug_Slip				:=	gs16_Sevcon1_Debug_Slip_Rx * SIXTEENTH_CF;
gr_Sevcon1_Debug_LmSat				:=	LREAL_TO_REAL(gs16_Sevcon1_Debug_LmSat_Rx * (1.52587890625 * EXPT(10, -5)));

END_PROGRAM

// Application/UserCode/CAN Function Blocks/CAN2/Receive_CAN2_EXD
FUNCTION_BLOCK Receive_CAN2_EXD
VAR_INPUT
	u32_COBID	:	DWORD;
END_VAR
VAR_OUTPUT
	q_NewData	:	BOOL;
	au8_Data	:	ARRAY [0..7] OF BYTE;
	u8_Length	:	BYTE;
END_VAR
VAR
	hq_Initialise	:	BOOL	:=	FALSE;
	ht_RxMessage	:	t_CANReceive;
	ht_MsgRx		:	Callback_Receive_CAN1;
END_VAR



IF (hq_Initialise = FALSE) THEN
	(*
	IF (u32_COBID > 16#7FF) THEN
		(*29 bit*)
		;
	ELSE
		(*11 bit*)
		;
	END_IF
	*)
	(*
	(*11 bit*)
	G_CAN2_Channel.AddCOBID(i_CobId := u32_COBID,
							i_itfCallback := ht_RxMessage,
							i_Argument := ADR(ht_RxMessage));
	*)
	(*29 bit*)
	G_CAN2_Channel.AddCOBID(i_CobId := u32_COBID OR EPEC_CANVXD.MASK_29BIT,
							i_itfCallback := ht_MsgRx,
							i_Argument := ADR(ht_RxMessage));
	(*G_CAN2_Channel.SetMask(i_CobID := u32_COBID OR EPEC_CANVXD.MASK_29BIT, i_Mask := 16#0C009000 OR EPEC_CANVXD.MASK_29BIT);
*)
	hq_Initialise	:=	TRUE;
END_IF


IF (ht_RxMessage.q_NewDataRxed = TRUE) THEN
	au8_Data	:=	ht_RxMessage.Data;
	u8_Length	:=	ht_RxMessage.Len;
	q_NewData	:=	TRUE;
	ht_RxMessage.q_NewDataRxed	:=	FALSE;
ELSE
	q_NewData	:=	FALSE;
END_IF

END_FUNCTION_BLOCK

// Application/UserCode/Sevcon_Compressor/Sevcon2_Rx
PROGRAM Sevcon2_Rx
VAR
	Compressor_Oil_Rx	:	Receive_CAN2_EXD;
	Compressor_Temp_Rx	:	Receive_CAN2_STD;
	TorqueStatus1_Rx	:	Receive_CAN2_EXD;
	TorqueStatus2_Rx	:	Receive_CAN2_EXD;
	TempStatus_Rx		:	Receive_CAN2_EXD;
	FaultStatus_Rx		:	Receive_CAN2_EXD;
	EncoderStatus_Rx	:	Receive_CAN2_EXD;
	DeubgCurrents_Rx	:	Receive_CAN2_EXD;
	DebugTemps1_Rx		:	Receive_CAN2_EXD;
	DebugTemps2_Rx		:	Receive_CAN2_EXD;
	DebugPMACControl_Rx	:	Receive_CAN2_EXD;
	DebugFVControl_Rx	:	Receive_CAN2_EXD;
	
	TorqueStatus1_Rx_Timer		:	TON;
	TorqueStatus2_Rx_Timer		:	TON;
	TempStatus_Rx_Timer			:	TON;
	FaultStatus_Rx_Timer		:	TON;
	EncoderStatus_Rx_Timer		:	TON;
	DeubgCurrents_Rx_Timer		:	TON;
	DebugTemps1_Rx_Timer		:	TON;
	DebugTemps2_Rx_Timer		:	TON;
	DebugPMACControl_Rx_Timer	:	TON;
	DebugFVControl_Rx_Timer		:	TON;
	Compressor_Temperature		: 	INT;
	Compressor_Oil_Switch		:	BYTE;
	
END_VAR

Compressor_Oil_Rx(u32_COBID	:=	16#1948FF72,
				q_NewData => ,
				au8_Data => ,
				u8_Length => 			);

Compressor_Temp_Rx(u32_COBID	:=	16#443,
				q_NewData => ,
				au8_Data => ,
				u8_Length => 			);

TorqueStatus1_Rx(u32_COBID	:=	16#1918FF72,
				q_NewData => ,
				au8_Data => ,
				u8_Length => 			);

TorqueStatus2_Rx(u32_COBID	:=	16#1919FF72,
				q_NewData => ,
				au8_Data => ,
				u8_Length => 			);

TempStatus_Rx(u32_COBID	:=	16#191AFF72,
				q_NewData => ,
				au8_Data => ,
				u8_Length => 			);

FaultStatus_Rx(u32_COBID	:=	16#191BFF72,
				q_NewData => ,
				au8_Data => ,
				u8_Length => 			);

EncoderStatus_Rx(u32_COBID	:=	16#191CFF72,
				q_NewData => ,
				au8_Data => ,
				u8_Length => 			);

DeubgCurrents_Rx(u32_COBID	:=	16#1928FF72,
				q_NewData => ,
				au8_Data => ,
				u8_Length => 			);

DebugTemps1_Rx(u32_COBID	:=	16#192AFF72,
				q_NewData => ,
				au8_Data => ,
				u8_Length => 			);

DebugTemps2_Rx(u32_COBID	:=	16#192BFF72,
				q_NewData => ,
				au8_Data => ,
				u8_Length => 			);

DebugPMACControl_Rx(u32_COBID	:=	16#192CFF72,
				q_NewData => ,
				au8_Data => ,
				u8_Length => 			);

DebugFVControl_Rx(u32_COBID	:=	16#192DFF72,
				q_NewData => ,
				au8_Data => ,
				u8_Length => 			);				

Compressor_Oil_Switch					:=	BIT_TO_BYTE (Compressor_Oil_Rx.au8_Data[2].4) +
											BIT_TO_BYTE (Compressor_Oil_Rx.au8_Data[2].5);

Compressor_Temperature					:=	Compressor_Temp_Rx.au8_Data[5] +
											Compressor_Temp_Rx.au8_Data[6];
				
gs16_Sevcon2_TorqueMeasured_Rx			:=	USINT_TO_INT(TorqueStatus1_Rx.au8_Data[0]) +
											SHL(USINT_TO_INT(TorqueStatus1_Rx.au8_Data[1]), 8);
gs16_Sevcon2_SpeedMeasured				:=	USINT_TO_INT(TorqueStatus1_Rx.au8_Data[2]) +
											SHL(USINT_TO_INT(TorqueStatus1_Rx.au8_Data[3]), 8);
gs16_Sevcon2_DCLink_Current				:=	USINT_TO_INT(TorqueStatus1_Rx.au8_Data[4]) +
											SHL(USINT_TO_INT(TorqueStatus1_Rx.au8_Data[5]), 8);
gu8_Sevcon2_SEQ_Torque					:=	TorqueStatus1_Rx.au8_Data[6];
gu8_Sevcon2_CS_Torque					:=	TorqueStatus1_Rx.au8_Data[7];

gs16_Sevcon2_TorqueAvailableForward_Rx	:=	USINT_TO_INT(TorqueStatus2_Rx.au8_Data[0]) +
											SHL(USINT_TO_INT(TorqueStatus2_Rx.au8_Data[1]), 8);
gs16_Sevcon2_TorqueAvailableReverse_Rx	:=	USINT_TO_INT(TorqueStatus2_Rx.au8_Data[2]) +
											SHL(USINT_TO_INT(TorqueStatus2_Rx.au8_Data[3]), 8);
gu8_Sevcon2_InverterStatus				:=	TorqueStatus2_Rx.au8_Data[4];
gu8_Sevcon2_TorqueLimitCode				:=	TorqueStatus2_Rx.au8_Data[5];
gu8_Sevcon2_SEQ_Status					:=	TorqueStatus2_Rx.au8_Data[6];
gu8_Sevcon2_CS_Status					:=	TorqueStatus2_Rx.au8_Data[7];

gs16_Sevcon2_TempRemaining				:=	USINT_TO_INT(TempStatus_Rx.au8_Data[0]) +
											SHL(USINT_TO_INT(TempStatus_Rx.au8_Data[1]), 8);
gs16_Sevcon2_MotorTemp					:=	USINT_TO_INT(TempStatus_Rx.au8_Data[2]) +
											SHL(USINT_TO_INT(TempStatus_Rx.au8_Data[3]), 8);
gs16_Sevcon2_DCLink_Voltage_Rx			:=	USINT_TO_INT(TempStatus_Rx.au8_Data[4]) +
											SHL(USINT_TO_INT(TempStatus_Rx.au8_Data[5]), 8);
gu8_Sevcon2_SEQ_Temp					:=	TempStatus_Rx.au8_Data[6];
gu8_Sevcon2_CS_Temp						:=	TempStatus_Rx.au8_Data[7];

gs16_Sevcon2_FaultCode					:=	USINT_TO_INT(FaultStatus_Rx.au8_Data[0]) +
											SHL(USINT_TO_INT(FaultStatus_Rx.au8_Data[1]), 8);
gs32_Sevcon2_FaultData					:=	USINT_TO_DINT(FaultStatus_Rx.au8_Data[2]) +
											SHL(USINT_TO_DINT(FaultStatus_Rx.au8_Data[3]), 8) +
											SHL(USINT_TO_DINT(FaultStatus_Rx.au8_Data[4]), 16) +
											SHL(USINT_TO_DINT(FaultStatus_Rx.au8_Data[5]), 24);
gu8_Sevcon2_SEQ_Fault					:=	FaultStatus_Rx.au8_Data[6];
gu8_Sevcon2_CS_Fault					:=	FaultStatus_Rx.au8_Data[7];

gs32_Sevcon2_EncoderPosition_Rx			:=	USINT_TO_DINT(EncoderStatus_Rx.au8_Data[0]) +
											SHL(USINT_TO_DINT(EncoderStatus_Rx.au8_Data[1]), 8) +
											SHL(USINT_TO_DINT(EncoderStatus_Rx.au8_Data[2]), 16) +
											SHL(USINT_TO_DINT(EncoderStatus_Rx.au8_Data[3]), 24);

gs16_Sevcon2_Debug_Id_Act_Rx			:=	USINT_TO_INT(DeubgCurrents_Rx.au8_Data[0]) +
											SHL(USINT_TO_INT(DeubgCurrents_Rx.au8_Data[1]), 8);
gs16_Sevcon2_Debug_Iq_Act_Rx			:=	USINT_TO_INT(DeubgCurrents_Rx.au8_Data[2]) +
											SHL(USINT_TO_INT(DeubgCurrents_Rx.au8_Data[3]), 8);
gs16_Sevcon2_Debug_Id_Ref_Rx			:=	USINT_TO_INT(DeubgCurrents_Rx.au8_Data[4]) +
											SHL(USINT_TO_INT(DeubgCurrents_Rx.au8_Data[5]), 8);
gs16_Sevcon2_Debug_Iq_Ref_Rx			:=	USINT_TO_INT(DeubgCurrents_Rx.au8_Data[6]) +
											SHL(USINT_TO_INT(DeubgCurrents_Rx.au8_Data[7]), 8);

gu8_Sevcon2_Debug_Temp_Junction0		:=	DebugTemps1_Rx.au8_Data[0];
gu8_Sevcon2_Debug_Temp_Junction1		:=	DebugTemps1_Rx.au8_Data[1];
gu8_Sevcon2_Debug_Temp_Junction2		:=	DebugTemps1_Rx.au8_Data[2];
gu8_Sevcon2_Debug_Temp_Junction3		:=	DebugTemps1_Rx.au8_Data[3];
gu8_Sevcon2_Debug_Temp_Junction4		:=	DebugTemps1_Rx.au8_Data[4];
gu8_Sevcon2_Debug_Temp_Junction5		:=	DebugTemps1_Rx.au8_Data[5];
gu8_Sevcon2_Debug_Temp_MotorMeasured	:=	DebugTemps1_Rx.au8_Data[6];
gu8_Sevcon2_Debug_Temp_MotorEstimate	:=	DebugTemps1_Rx.au8_Data[7];

gu8_Sevcon2_Debug_Temp_CapEstimateFast	:=	DebugTemps2_Rx.au8_Data[0];
gu8_Sevcon2_Debug_Temp_Track			:=	DebugTemps2_Rx.au8_Data[1];
gu8_Sevcon2_Debug_Temp_CapEstimateSlow	:=	DebugTemps2_Rx.au8_Data[2];
gu8_Sevcon2_Debug_Temp_Heatsink			:=	DebugTemps2_Rx.au8_Data[3];
gu8_Sevcon2_Debug_Temp_DeltaTj			:=	DebugTemps2_Rx.au8_Data[4];
gu8_Sevcon2_Debug_Temp_Normalised		:=	DebugTemps2_Rx.au8_Data[5];
gu8_Sevcon2_Debug_Temp_Coolant			:=	DebugTemps2_Rx.au8_Data[6];
gu8_Sevcon2_Debug_Temp_Winding			:=	DebugTemps2_Rx.au8_Data[7];

gs16_Sevcon2_Debug_MaxFlux				:=	USINT_TO_INT(DebugPMACControl_Rx.au8_Data[0]) +
											SHL(USINT_TO_INT(DebugPMACControl_Rx.au8_Data[1]), 8);
gs16_Sevcon2_Debug_IvLim				:=	USINT_TO_INT(DebugPMACControl_Rx.au8_Data[2]) +
											SHL(USINT_TO_INT(DebugPMACControl_Rx.au8_Data[3]), 8);
gs16_Sevcon2_Debug_IqMax				:=	USINT_TO_INT(DebugPMACControl_Rx.au8_Data[4]) +
											SHL(USINT_TO_INT(DebugPMACControl_Rx.au8_Data[5]), 8);
gs16_Sevcon2_Debug_Ls_Rx				:=	USINT_TO_INT(DebugPMACControl_Rx.au8_Data[6]) +
											SHL(USINT_TO_INT(DebugPMACControl_Rx.au8_Data[7]), 8);

gs16_Sevcon2_Debug_Slip_Rx				:=	USINT_TO_INT(DebugFVControl_Rx.au8_Data[0]) +
											SHL(USINT_TO_INT(DebugFVControl_Rx.au8_Data[1]), 8);
gs16_Sevcon2_Debug_LmSat_Rx				:=	USINT_TO_INT(DebugFVControl_Rx.au8_Data[2]) +
											SHL(USINT_TO_INT(DebugFVControl_Rx.au8_Data[3]), 8);
gs16_Sevcon2_Debug_IqMax2				:=	USINT_TO_INT(DebugFVControl_Rx.au8_Data[4]) +
											SHL(USINT_TO_INT(DebugFVControl_Rx.au8_Data[5]), 8);
gs16_Sevcon2_Debug_RecipFlux			:=	USINT_TO_INT(DebugFVControl_Rx.au8_Data[6]) +
											SHL(USINT_TO_INT(DebugFVControl_Rx.au8_Data[7]), 8);

											
TorqueStatus1_Rx_Timer(IN := NOT(TorqueStatus1_Rx.q_NewData), PT := T#3S);
TorqueStatus2_Rx_Timer(IN := NOT(TorqueStatus2_Rx.q_NewData), PT := T#3S);
TempStatus_Rx_Timer(IN := NOT(TempStatus_Rx.q_NewData), PT := T#3S);
FaultStatus_Rx_Timer(IN := NOT(FaultStatus_Rx.q_NewData), PT := T#3S);
EncoderStatus_Rx_Timer(IN := NOT(EncoderStatus_Rx.q_NewData), PT := T#3S);
DeubgCurrents_Rx_Timer(IN := NOT(DeubgCurrents_Rx.q_NewData), PT := T#3S);
DebugTemps1_Rx_Timer(IN := NOT(DebugTemps1_Rx.q_NewData), PT := T#3S);
DebugTemps2_Rx_Timer(IN := NOT(DebugTemps2_Rx.q_NewData), PT := T#3S);
DebugPMACControl_Rx_Timer(IN := NOT(DebugPMACControl_Rx.q_NewData), PT := T#3S);
DebugFVControl_Rx_Timer(IN := NOT(DebugFVControl_Rx.q_NewData), PT := T#3S);
IF (TorqueStatus1_Rx_Timer.Q = TRUE AND TorqueStatus2_Rx_Timer.Q = TRUE AND TempStatus_Rx_Timer.Q = TRUE AND
	FaultStatus_Rx_Timer.Q = TRUE AND EncoderStatus_Rx_Timer.Q = TRUE AND DeubgCurrents_Rx_Timer.Q = TRUE AND
	DebugTemps1_Rx_Timer.Q = TRUE AND DebugTemps2_Rx_Timer.Q = TRUE AND DebugPMACControl_Rx_Timer.Q = TRUE AND
	DebugFVControl_Rx_Timer.Q = TRUE) THEN
	gq_Sevcon2_CommsLoss	:=	TRUE;
ELSE
	gq_Sevcon2_CommsLoss	:=	FALSE;
END_IF											


Sevcon2_RxConversion();

END_PROGRAM

// Application/UserCode/Sevcon_Compressor/Sevcon2_RxConversion
PROGRAM Sevcon2_RxConversion
VAR
END_VAR
VAR CONSTANT
	SIXTEENTH_CF	:	REAL	:=	0.0625;
END_VAR




gr_Sevcon2_TorqueMeasured			:=	gs16_Sevcon2_TorqueMeasured_Rx * SIXTEENTH_CF;
gr_Sevcon2_TorqueAvailableForward	:=	gs16_Sevcon2_TorqueAvailableForward_Rx * SIXTEENTH_CF;
gr_Sevcon2_TorqueAvailableReverse	:=	gs16_Sevcon2_TorqueAvailableReverse_Rx * SIXTEENTH_CF;
gr_Sevcon2_DCLink_Voltage			:=	gs16_Sevcon2_DCLink_Voltage_Rx * SIXTEENTH_CF;
gr_Sevcon2_EncoderPosition			:=	LREAL_TO_REAL(gs32_Sevcon2_EncoderPosition_Rx * (1.5287890625 * EXPT(10, -5)));
gr_Sevcon2_Debug_Id_Act				:=	gs16_Sevcon2_Debug_Id_Act_Rx * SIXTEENTH_CF;
gr_Sevcon2_Debug_Iq_Act				:=	gs16_Sevcon2_Debug_Iq_Act_Rx * SIXTEENTH_CF;
gr_Sevcon2_Debug_Id_Ref				:=	gs16_Sevcon2_Debug_Id_Ref_Rx * SIXTEENTH_CF;
gr_Sevcon2_Debug_Iq_Ref				:=	gs16_Sevcon2_Debug_Iq_Ref_Rx * SIXTEENTH_CF;
gr_Sevcon2_Debug_Ls					:=	LREAL_TO_REAL(gs16_Sevcon2_Debug_Ls_Rx * (5.960464477539 * EXPT(10, -8)));
gr_Sevcon2_Debug_Slip				:=	gs16_Sevcon2_Debug_Slip_Rx * SIXTEENTH_CF;
gr_Sevcon2_Debug_LmSat				:=	LREAL_TO_REAL(gs16_Sevcon2_Debug_LmSat_Rx * (1.52587890625 * EXPT(10, -5)));

END_PROGRAM

// Application/UserCode/CAN Function Blocks/CAN2/Receive_CAN2_STD
FUNCTION_BLOCK Receive_CAN2_STD
VAR_INPUT
	u32_COBID	:	DWORD;
END_VAR
VAR_OUTPUT
	q_NewData	:	BOOL;
	au8_Data	:	ARRAY [0..7] OF BYTE;
	u8_Length	:	BYTE;
END_VAR
VAR
	hq_Initialise	:	BOOL	:=	FALSE;
	ht_RxMessage	:	t_CANReceive;
	ht_MsgRx		:	Callback_Receive_CAN1;
END_VAR



IF (hq_Initialise = FALSE) THEN
	(*
	IF (u32_COBID > 16#7FF) THEN
		(*29 bit*)
		;
	ELSE
		(*11 bit*)
		;
	END_IF
	*)
	
	(*11 bit*)
	G_CAN2_Channel.AddCOBID(i_CobId := u32_COBID,
							i_itfCallback := ht_MsgRx,
							i_Argument := ADR(ht_RxMessage));
	(*
	(*29 bit*)
	G_CAN2_Channel.AddCOBID(i_CobId := u32_COBID OR EPEC_CANVXD.MASK_29BIT,
							i_itfCallback := ht_MsgRx,
							i_Argument := ADR(ht_RxMessage));
*)	(*G_CAN2_Channel.SetMask(i_CobID := u32_COBID OR EPEC_CANVXD.MASK_29BIT, i_Mask := 16#0C009000 OR EPEC_CANVXD.MASK_29BIT);
*)
	hq_Initialise	:=	TRUE;
END_IF


IF (ht_RxMessage.q_NewDataRxed = TRUE) THEN
	au8_Data	:=	ht_RxMessage.Data;
	u8_Length	:=	ht_RxMessage.Len;
	q_NewData	:=	TRUE;
	ht_RxMessage.q_NewDataRxed	:=	FALSE;
ELSE
	q_NewData	:=	FALSE;
END_IF

END_FUNCTION_BLOCK

// Application/UserCode/Brusa/Brusa1_Comms/Brusa1_Rx
PROGRAM Brusa1_Rx
VAR
	ActAC_Rx			:	Receive_CAN2_STD;
	ActErr_Rx			:	Receive_CAN2_STD;
	ActInt_Rx			:	Receive_CAN2_STD;
	ActLim_Rx			:	Receive_CAN2_STD;
	ActPlug_Rx			:	Receive_CAN2_STD;
	
	ActAC_Rx_Timer		:	TON;
	ActErr_Rx_Timer		:	TON;
	ActInt_Rx_Timer		:	TON;
	ActLim_Rx_Timer		:	TON;
	ActPlug_Rx_Timer	:	TON;
	
	StatusPP_Rx			:	USINT; 
	StatusPP_Prev		:	USINT;
	
	ACVoltL1Act_Rx		:	USINT;
	ACVoltL2Act_Rx		:	USINT;
	ACVoltL3Act_Rx		:	USINT;
	ACFreqAct			:	USINT;
	SACPhaseRot			:	BOOL;
	ACCurrL1Act_Rx		:	USINT;
	ACCurrL2Act_Rx		:	USINT;
	ACCurrL3Act_Rx		:	USINT;
	ACPowTotAct_Rx		:	USINT;
	
	(*Act Err*)
	E_WrongHW			: BOOL;
	E_WrongFPGA			: BOOL;
	E_EPGAInit			: BOOL;
	E_NVSRam			: BOOL;
	E_Flash				: BOOL;
	E_OSTrap			: BOOL;
	E_HVIsoPos			: BOOL;
	E_HVIsoNeg			: BOOL;
	E_Internal			: BOOL;
	E_TempInt			: BOOL;
	E_DCHVVoltRed		: BOOL;
	E_IntSupply			: BOOL;
	E_CANMsgLost		: BOOL;
	E_CANValue			: BOOL;
	E_ACInterruption	: BOOL;
	E_DCHVVoltRange		: BOOL;
	E_TempCon			: BOOL;
	E_ConLocked			: BOOL;
	E_Interlock			: BOOL;
	E_Crash				: BOOL;
	E_PRELOAD			: BOOL;
	E_BURST				: BOOL;
	E_TPON				: BOOL;
	E_UZK				: BOOL;
	E_LatchFPGA			: BOOL;
	E_OverTemp			: BOOL;
	(*Warnings*)
	W_Watchdog			: BOOL;
	W_PowRed			: BOOL;
	W_TempInt			: BOOL;
	W_CANTimeout		: BOOL;
	W_CANOff			: BOOL;
	W_CANRx				: BOOL;
	W_CANTx				: BOOL;
	W_ConLocked			: BOOL;
	W_FPGA				: BOOL;
	W_ACVoltage			: BOOL;
	W_ACFrequency		: BOOL;
	W_PRELOAD			: BOOL;
	
	(*Act Int*)
	ACWhAct				:	UINT;
	DCHVWhAct			:	UINT;
	MaxTempAct_Rx		:	USINT;
	TempCon_Rx			:	USINT;
	DCHVAhAct_Rx		:	UINT;
	(*Act Lim*)
	StateCrtlPilot		:	USINT;
	DCHVVoltAct_Rx		:	UINT;
	StateAct			:	USINT; //0:Sleep 1:Wakeup 2:Standby 3:Ready2Charge 4:Charge 5:Shutdown
	S_DCHVCurrLim		:	BOOL;
	S_DCHVVoltLim		:	BOOL;
	DCHVCurrAct_Rx		:	UINT;
	S_ProximityLim		:	BOOL;
	S_CtrlPilotLim		:	BOOL;
	S_ConTempLim		:	BOOL;
	S_IntTempLim		:	BOOL;
	S_ACCurrLim			:	BOOL;
	ACCurrMaxAct_Rx		:	UINT;
	ACCurrHWAvl_Rx		:	USINT;
	S_ProximityDet		:	BOOL;
	S_CtrlPilotDet		:	BOOL;
	S_ConLocked			:	BOOL;
	S_ACDet				:	BOOL;
	S_HWWakeup			:	BOOL;
	S_HWEnablErre		:	BOOL;
	S_Err				:	BOOL;
	S_Warn				:	BOOL;
	(*Act Plug*)
	StatusCP			:	USINT;
	S_CPX1				:	BOOL;
	S_CPSCC				:	BOOL;
	ACCurrMaxCP_Rx		:	UINT;
	StatusPP			:	USINT; //0:PROXD_DETECTED 1:PROXD_CIRCUIT_RANGE 2:PROXD_CIRCUIT_LOW 3:PROXD_CIRCUIT_HIGH 4:PROXD_CIRCUIT_ERRATIC 5:PROXD_NOT_CONNECTED 7:SNA
	ACCurrMaxPP			:	USINT; //0:0 A 1:13 A 2:20 A 3:32 A 4:63 A 7:SNA
	s_ACVoltDerate		:	BOOL;
	S_ACDerating		:	BOOL;
	ACPhaseUsd			:	USINT;
	ACPhaseDet			:	USINT;  ///kak Why not used?????????
	CoolingRequest		:	USINT;
	TempCoolPlate_Rx	:	USINT; //Actual temperatur cool plate 255:SNA
	CommsLoss			:	BOOL;
	C_EnPhaseShift		:	BOOL;
END_VAR


ActAC_Rx(u32_COBID	:=	16#729,
				q_NewData => ,
				au8_Data => ,
				u8_Length => 			);
				
ActErr_Rx(u32_COBID	:=	16#799,
				q_NewData => ,
				au8_Data => ,
				u8_Length => 			);
				
ActInt_Rx(u32_COBID	:=	16#709,
				q_NewData => ,
				au8_Data => ,
				u8_Length => 			);
				
ActLim_Rx(u32_COBID	:=	16#728,
				q_NewData => ,
				au8_Data => ,
				u8_Length => 			);
				
ActPlug_Rx(u32_COBID	:=	16#739,
				q_NewData => ,
				au8_Data => ,
				u8_Length => 			);

(*Act AC*)
ACVoltL1Act_Rx		:=	ActAC_Rx.au8_Data[0];
ACVoltL2Act_Rx		:=	ActAC_Rx.au8_Data[1];
ACVoltL3Act_Rx		:=	ActAC_Rx.au8_Data[2];
ACFreqAct			:=	(ActAC_Rx.au8_Data[3] AND 2#01111111); (*Mask*)
SACPhaseRot			:=	ActAC_Rx.au8_Data[3].7;
ACCurrL1Act_Rx		:=	ActAC_Rx.au8_Data[4];
ACCurrL2Act_Rx		:=	ActAC_Rx.au8_Data[5];
ACCurrL3Act_Rx		:=	ActAC_Rx.au8_Data[6];
ACPowTotAct_Rx		:=	ActAC_Rx.au8_Data[7];;

(*Act Err*)
E_WrongHW			:=	ActErr_Rx.au8_Data[0].0;
E_WrongFPGA			:=	ActErr_Rx.au8_Data[0].1;
E_EPGAInit			:=	ActErr_Rx.au8_Data[0].2;
E_NVSRam			:=	ActErr_Rx.au8_Data[0].5;
E_Flash				:=	ActErr_Rx.au8_Data[0].6;
E_OSTrap			:=	ActErr_Rx.au8_Data[0].7;
E_HVIsoPos			:=	ActErr_Rx.au8_Data[1].1;
E_HVIsoNeg			:=	ActErr_Rx.au8_Data[1].2;
E_Internal			:=	ActErr_Rx.au8_Data[1].4;
E_TempInt			:=	ActErr_Rx.au8_Data[1].5;
E_DCHVVoltRed		:=	ActErr_Rx.au8_Data[1].6;
E_IntSupply			:=	ActErr_Rx.au8_Data[1].7;
E_CANMsgLost		:=	ActErr_Rx.au8_Data[2].0;
E_CANValue			:=	ActErr_Rx.au8_Data[2].1;
E_ACInterruption	:=	ActErr_Rx.au8_Data[2].2;
E_DCHVVoltRange		:=	ActErr_Rx.au8_Data[2].3;
E_TempCon			:=	ActErr_Rx.au8_Data[2].4;
E_ConLocked			:=	ActErr_Rx.au8_Data[2].5;
E_Interlock			:=	ActErr_Rx.au8_Data[2].6;
E_Crash				:=	ActErr_Rx.au8_Data[2].7;
E_PRELOAD			:=	ActErr_Rx.au8_Data[3].1;
E_BURST				:=	ActErr_Rx.au8_Data[3].2;
E_TPON				:=	ActErr_Rx.au8_Data[3].3;
E_UZK				:=	ActErr_Rx.au8_Data[3].4;
E_LatchFPGA			:=	ActErr_Rx.au8_Data[3].5;
E_OverTemp			:=	ActErr_Rx.au8_Data[3].7;
W_Watchdog			:=	ActErr_Rx.au8_Data[4].7;
W_PowRed			:=	ActErr_Rx.au8_Data[5].0;
W_TempInt			:=	ActErr_Rx.au8_Data[5].1;
W_CANTimeout		:=	ActErr_Rx.au8_Data[6].0;
W_CANOff			:=	ActErr_Rx.au8_Data[6].1;
W_CANRx				:=	ActErr_Rx.au8_Data[6].2;
W_CANTx				:=	ActErr_Rx.au8_Data[6].3;
W_ConLocked			:=	ActErr_Rx.au8_Data[6].7;
W_FPGA				:=	ActErr_Rx.au8_Data[7].0;
W_ACVoltage			:=	ActErr_Rx.au8_Data[7].1;
W_ACFrequency		:=	ActErr_Rx.au8_Data[7].2;
W_PRELOAD			:=	ActErr_Rx.au8_Data[7].3;


(*Act Int*)
ACWhAct			:=	SHL(USINT_TO_UINT(ActInt_Rx.au8_Data[0]), 8) +
								USINT_TO_UINT(ActInt_Rx.au8_Data[1]);
DCHVWhAct			:=	SHL(USINT_TO_UINT(ActInt_Rx.au8_Data[2]), 8) +
								USINT_TO_UINT(ActInt_Rx.au8_Data[3]);
MaxTempAct_Rx		:=	ActInt_Rx.au8_Data[4];
TempCon_Rx			:=	ActInt_Rx.au8_Data[5];
DCHVAhAct_Rx		:=	SHL(USINT_TO_UINT(ActInt_Rx.au8_Data[6]), 8) +
								USINT_TO_UINT(ActInt_Rx.au8_Data[7]);
(*Act Lim*)
StateCrtlPilot		:=	SHR((ActLim_Rx.au8_Data[0] AND 2#11100000), 5);
DCHVVoltAct_Rx	:=	SHL(USINT_TO_UINT(ActLim_Rx.au8_Data[0] AND 2#00011111), 8) +
								USINT_TO_UINT(ActLim_Rx.au8_Data[1]);
StateAct			:=	SHR((ActLim_Rx.au8_Data[2] AND 2#11100000), 5);
S_DCHVCurrLim		:=	ActLim_Rx.au8_Data[2].4;
S_DCHVVoltLim		:=	ActLim_Rx.au8_Data[2].3;
DCHVCurrAct_Rx	:=	SHL(USINT_TO_UINT(ActLim_Rx.au8_Data[2] AND 2#00000111), 8) +
								USINT_TO_UINT(ActLim_Rx.au8_Data[3]);
S_ProximityLim		:=	ActLim_Rx.au8_Data[4].7;
S_CtrlPilotLim		:=	ActLim_Rx.au8_Data[4].6;
S_ConTempLim		:=	ActLim_Rx.au8_Data[4].5;
S_IntTempLim		:=	ActLim_Rx.au8_Data[4].4;
S_ACCurrLim			:=	ActLim_Rx.au8_Data[4].3;
ACCurrMaxAct_Rx	:=	SHL(USINT_TO_UINT(ActLim_Rx.au8_Data[4] AND 2#00000111), 8) +
								USINT_TO_UINT(ActLim_Rx.au8_Data[5]);
ACCurrHWAvl_Rx		:=	ActLim_Rx.au8_Data[6];
S_ProximityDet		:=	ActLim_Rx.au8_Data[7].7;
S_CtrlPilotDet		:=	ActLim_Rx.au8_Data[7].6;
S_ConLocked			:=	ActLim_Rx.au8_Data[7].5;
S_ACDet				:=	ActLim_Rx.au8_Data[7].4;
S_HWWakeup			:=	ActLim_Rx.au8_Data[7].3;
S_HWEnablErre		:=	ActLim_Rx.au8_Data[7].2;
S_Err				:=	ActLim_Rx.au8_Data[7].1;
S_Warn				:=	ActLim_Rx.au8_Data[7].0;
(*Act Plug*)
StatusCP			:=	ActPlug_Rx.au8_Data[0] AND 2#11100000;
S_CPX1				:=	ActPlug_Rx.au8_Data[0].4;
S_CPSCC				:=	ActPlug_Rx.au8_Data[0].3;
ACCurrMaxCP_Rx	:=	SHL(USINT_TO_UINT(ActPlug_Rx.au8_Data[0] AND 2#00000011), 8) +
								USINT_TO_UINT(ActPlug_Rx.au8_Data[1]);
StatusPP_Rx			:=	SHR((ActPlug_Rx.au8_Data[2] AND 2#01110000), 4);
ACCurrMaxPP		:=	ActPlug_Rx.au8_Data[2] AND 2#00001111;
s_ACVoltDerate		:=	ActPlug_Rx.au8_Data[4].7;
S_ACDerating		:=	ActPlug_Rx.au8_Data[4].6;
ACPhaseUsd			:=	SHR((ActPlug_Rx.au8_Data[4] AND 2#00111000), 3);
ACPhaseDet			:=	ActPlug_Rx.au8_Data[4] AND 2#00000111;
CoolingRequest		:=	ActPlug_Rx.au8_Data[5] AND 2#01111111;
TempCoolPlate_Rx	:=	ActPlug_Rx.au8_Data[6];


IF NOT(Brusa1_Tx.hton_NoPP_StopTx_Timer.Q) THEN
	ActAC_Rx_Timer(IN := NOT(ActAC_Rx.q_NewData), PT := T#5S);
	ActErr_Rx_Timer(IN := NOT(ActErr_Rx.q_NewData), PT := T#5S);
	ActInt_Rx_Timer(IN := NOT(ActInt_Rx.q_NewData), PT := T#5S);
	ActLim_Rx_Timer(IN := NOT(ActLim_Rx.q_NewData), PT := T#5S);
	ActPlug_Rx_Timer(IN := NOT(ActPlug_Rx.q_NewData), PT := T#5S);
	
	IF (ActAC_Rx_Timer.Q AND ActErr_Rx_Timer.Q AND ActInt_Rx_Timer.Q AND
		ActLim_Rx_Timer.Q AND ActPlug_Rx_Timer.Q) THEN
		CommsLoss	:=	TRUE;
	ELSE
		CommsLoss	:=	FALSE;
	END_IF
END_IF

(*Only update Status PP if both this value and the previous value are the same*)
IF (StatusPP_Rx = StatusPP_Prev) THEN
	StatusPP	:=	StatusPP_Rx;
END_IF
StatusPP_Prev	:=	StatusPP_Rx;

Brusa1_RxConversion();

END_PROGRAM

// Application/UserCode/Brusa/Brusa1_Comms/Brusa1_Tx
PROGRAM Brusa1_Tx
VAR
	DenLim_Tx				:	EPEC_CANVXD.Msg;
	hu8_DenLim_Tx0			:	BYTE;
	hu8_DenLim_Tx2			:	BYTE;
	hu8_DenLim_Tx4			:	BYTE;
	hu8_DenLim_Tx6			:	BYTE;
	hton_Transmit_Timer		:	TON;
	hton_NoPP_StopTx_Timer	:	TON;
	StopBroadcast			:	BOOL;
	C_VentilRq				: 	BOOL;
END_VAR

//r2

Brusa1_TxConversion();

StopBroadcast	:=	(NOT(Brusa1_Rx.S_ProximityDet)(* AND DI_q_VehicleKL15_DI = FALSE*));
hton_NoPP_StopTx_Timer(IN := StopBroadcast, PT := T#1S);

// Brusa1_Control.C_Clr_Err	:= FALSE; 

hu8_DenLim_Tx0	        :=	UINT_TO_USINT(SHR(Brusa1_TxConversion.DCHVVoltLimMax_Tx, 8)) + SHL(BOOL_TO_USINT(C_VentilRq), 5) +
					        SHL(BOOL_TO_USINT(Brusa.M_Unlock), 6) + SHL(BOOL_TO_USINT((*Brusa.M_ErrCLr*) FALSE), 7);
hu8_DenLim_Tx2	        :=	(UINT_TO_USINT(SHR(Brusa1_TxConversion.DCHVCurrLimMax_Tx, 8)) AND 2#00000111) + SHL(Brusa.M_StateDem, 5);
hu8_DenLim_Tx4	        :=	(UINT_TO_USINT(SHR(Brusa1_TxConversion.ACCurrLimMax_Tx, 8)) AND 2#00000111) + SHL(Brusa.LEDDem, 4);
//hu8_DenLim_Tx6	        :=	(UINT_TO_USINT(SHR(Brusa1_TxConversion.ACPhaseShift_Tx, 8)) AND 2#00001111) + SHL(BOOL_TO_USINT(Brusa1_Rx.C_EnPhaseShift), 4); //kak ac or en??????????????????????????

DenLim_Tx.ID		:=	16#711;
DenLim_Tx.Data[0]	:=	hu8_DenLim_Tx0;
DenLim_Tx.Data[1]	:=	UINT_TO_USINT(Brusa1_TxConversion.DCHVVoltLimMax_Tx);
DenLim_Tx.Data[2]	:=	hu8_DenLim_Tx2;
DenLim_Tx.Data[3]	:=	UINT_TO_USINT(Brusa1_TxConversion.DCHVCurrLimMax_Tx);
DenLim_Tx.Data[4]	:=	hu8_DenLim_Tx4;
DenLim_Tx.Data[5]	:=	UINT_TO_USINT(Brusa1_TxConversion.ACCurrLimMax_Tx);
DenLim_Tx.Data[6]	:=	hu8_DenLim_Tx6;
DenLim_Tx.Data[7]	:=	UINT_TO_USINT(Brusa1_TxConversion.ACPhaseShift_Tx);
DenLim_Tx.Len		:=	8;


hton_Transmit_Timer(IN := NOT(hton_Transmit_Timer.Q), PT := T#90MS);
IF (hton_Transmit_Timer.Q = TRUE AND NOT(hton_NoPP_StopTx_Timer.Q) = TRUE) THEN
	G_CAN2_Channel.SendMessage(i_pMSG:=ADR(DenLim_Tx));
END_IF

END_PROGRAM

// Application/UserCode/Brusa/Brusa1_Comms/Brusa1_TxConversion
PROGRAM Brusa1_TxConversion
VAR
		DCHVVoltLimMax_Tx	:	UINT;
		DCHVCurrLimMax_Tx	:	UINT;
		ACCurrLimMax_Tx		:	UINT;
		ACPhaseShift_Tx		:	UINT;
END_VAR


DCHVVoltLimMax_Tx	:=	REAL_TO_UINT(Brusa.M_DCHVVoltLimMax / 0.1);
DCHVCurrLimMax_Tx	:=	REAL_TO_UINT((Brusa.M_DCHVCurrLimMax - 102.4) / 0.1);
ACCurrLimMax_Tx		:=	REAL_TO_UINT((Brusa.M_ACCurrLimMax - 102.4) / 0.1);
//ACPhaseShift_Tx		:=	REAL_TO_UINT(Brusa1_Control.ACPhaseShift / 0.1);

END_PROGRAM

// Application/UserCode/Brusa/Brusa
(*==============================================================================================================*)
(*    Brusa charging function block calls and LED control                                                       *)
(*==============================================================================================================*)
PROGRAM Brusa
VAR
	Master           : BrusaControl; // Brusa charger master side
	Slave            : BrusaControl; // Brusa charger slave side
	
	LEDDem           : USINT; 
	LEDState         : BYTE;         // Case variable for LED states
	
	M_StateDem       : USINT;
	S_StateDem       : USINT;
	M_Unlock         : BOOL;
	S_Unlock         : BOOL;
	M_ErrCLr         : BOOL;
	S_ErrClr         : BOOL;
	M_ChargeStopAct  : BOOL;
	M_DCHVCurrLimMax : REAL;
	S_DCHVCurrLimMax : REAL;
	M_ACCurrLimMax   : REAL;
	S_ACCurrLimMax   : REAL;
	M_DCHVVoltLimMax : REAL;
	S_DCHVVoltLimMax : REAL;
	M_BalancingAmps  : REAL := 2;
	S_BalancingAmps  : REAL := 2;

	PulseTmr         : WORD;	
	PulseLength      : WORD := 50;    // Initialised to 500ms (50 * 10ms scans)
	Pulsing          : BOOL := FALSE;
	
	chargeStatus     : BYTE;
END_VAR
VAR CONSTANT
(*Charger statuswords =========================================================================================*)
	NLG_STATUS_CHARGE		: BYTE	:= 4;
	
(*Charger controlwords ========================================================================================*)
	NLG_CONTROL_STANDBY		: BYTE	:= 0;
	NLG_CONTROL_CHARGE		: BYTE	:= 1;
	
(*NLG LED States ==============================================================================================*)
	LED_OFF			        : BYTE	:= 0;
	LED_RED					: BYTE	:= 2;
	LED_GREEN_PULSE	        : BYTE  := 3;
	LED_GREEN				: BYTE	:= 4;
	LED_BLUE		        : BYTE	:= 8;
	LED_BLUE_GREEN_PULSE	: BYTE	:= 11;
	
(*Charge status  ==============================================================================================*)
	NOT_CONNECTED           : BYTE  := 0;
	STOPPED                 : BYTE  := 1;
	ERROR_ACTIVE            : BYTE  := 2;
	BALANCING               : BYTE  := 3;
	FULLY_CHARGED           : BYTE  := 4;
	NO_AC                   : BYTE  := 5;
	CHARGING                : BYTE  := 6;
	
END_VAR

(*==============================================================================================================*)
(*    Brusa charging function block calls                                                                       *)
(*==============================================================================================================*)
 // FreeContactor(); // Uncomment this to pulse welded contactors


Master (                Master := TRUE, // Master charger
	                 Safety_OK := OrionBMS2_RxConversion.Safety_OK,
                  CtrlPilotDet := Brusa1_Rx.S_CtrlPilotDet,
                  ProximityDet := Brusa1_Rx.S_ProximityDet,
                         Error := Brusa1_Rx.S_Err,
                         ACDet := Brusa1_Rx.S_ACDet,
               BalancingActive := gq_BMS1_BalActive,
                      SysState := gu8_SystemState,
                      StateAct := Brusa1_Rx.StateAct,
                        Status := Brusa1_Rx.StatusPP,
                Balancing_Amps := M_BalancingAmps,
         Offset_Charge_Voltage := 0,//(HMI_Rx.RAW_Pack_1_Offset_Volts   * 0.1),
                           CCL := gs16_BMS1_CCL,
		      MaxChargingVolts := gr_OrionBMS1_Max_Charging_Voltage,
			     StopChargeReq := HMI_Rx.StopChargeRq,
			 ReportedMaxACCurr := Brusa1_Rx.ACCurrMaxAct_Rx,
			         CPMaxAmps := Brusa1_Rx.ACCurrMaxCP_Rx,
						   
                      StateDem => M_StateDem,
				  StopCharging => ,
                        Unlock => M_Unlock,
                 ErrorClearOut => M_ErrCLr,
                DCHVCurrLimMax => M_DCHVCurrLimMax,
                  ACCurrLimMax => M_ACCurrLimMax,
                DCHVVoltLimMax => M_DCHVVoltLimMax );
						   
						   
Slave (                 Master := FALSE, // Slave charger
	                 Safety_OK := OrionBMS2_RxConversion.Safety_OK,
                  CtrlPilotDet := Brusa1_Rx.S_CtrlPilotDet,
                  ProximityDet := Brusa1_Rx.S_ProximityDet,
                         Error := Brusa2_Rx.S_Err,
                         ACDet := Brusa2_Rx.S_ACDet,
               BalancingActive := gq_BMS2_BalActive,
                      SysState := gu8_SystemState,
                      StateAct := Brusa2_Rx.StateAct,
                        Status := Brusa1_Rx.StatusPP,
                Balancing_Amps := S_BalancingAmps,
         Offset_Charge_Voltage := (HMI_Rx.RAW_Pack_2_Offset_Volts   * 0.1),
                           CCL := gs16_BMS2_CCL,
			  MaxChargingVolts := gr_OrionBMS1_Max_Charging_Voltage,
			     StopChargeReq := HMI_Rx.StopChargeRq,
             ReportedMaxACCurr := Brusa2_Rx.ACCurrMaxAct_Rx,
			 	     CPMaxAmps := Brusa1_Rx.ACCurrMaxCP_Rx,
						   
                      StateDem => S_StateDem,
                        //Unlock => S_Unlock,
                 ErrorClearOut => S_ErrCLr,
                DCHVCurrLimMax => S_DCHVCurrLimMax,
                  ACCurrLimMax => S_ACCurrLimMax,
                DCHVVoltLimMax => S_DCHVVoltLimMax);	

(*==============================================================================================================*)
(*    Brusa LED control                                                                                         *)
(*==============================================================================================================*)

// Check to see if the charger is plugged in
IF (gu8_SystemState = PLUGIN_SYS) THEN    
            
	// Check for any errors
	IF (gu8_SystemState = ERROR_SYS) THEN             
		LEDDem := LED_RED;
		chargeStatus := 1;
	
	// Check for fully charged
	ELSIF gq_BattFullyCharged THEN                                                       
		LEDDem := LED_GREEN;
	
	// Check to see if charging is active
	ELSIF ((Brusa1_Rx.StateAct = NLG_STATUS_CHARGE) OR (Brusa2_Rx.StateAct = NLG_STATUS_CHARGE)) THEN
		
		// Check to see if balancing is active (Only if charging is also active)
		IF (gq_BMS1_BalActive OR gq_BMS2_BalActive) THEN
			LEDDem := LED_BLUE_GREEN_PULSE;
		ELSE
			LEDDem := LED_BLUE;
		END_IF
		
	// Check to see that AC is detected
	ELSIF NOT (Brusa1_Rx.S_ACDet) THEN
		LEDDem := LED_GREEN_PULSE; 

END_IF

ELSE 
LEDDem := 0; // OFF 

END_IF

(*==============================================================================================================*)
(*    Charge status for HMI Tx                                                                                  *)
(*==============================================================================================================*)

// System is in error state
IF (gu8_SystemState = ERROR_SYS) THEN
	chargeStatus := ERROR_ACTIVE;

// System is in plug in state (charge plug detected)
ELSIF (gu8_SystemState = PLUGIN_SYS) THEN
	
	// Charge stopped by HMI
	IF (M_ChargeStopAct) THEN
		chargeStatus := STOPPED;
	
	// Vehicle is fully charged	
	ELSIF (BMSData.Batteries_Fully_Charged AND NOT (gq_BMS2_BalActive OR gq_BMS2_BalActive)) THEN
		chargeStatus := FULLY_CHARGED;
	
	// Waiting for AC	
	ELSIF NOT (Brusa1_Rx.S_ACDet AND Brusa2_Rx.S_ACDet) THEN
		chargeStatus := NO_AC; 
	
	// BMS is balancing	
	ELSIF (gq_BMS2_BalActive OR gq_BMS2_BalActive) THEN
		chargeStatus := BALANCING;
	
	// Vehicle is charging	
	ELSIF ((Brusa1_Rx.StateAct = NLG_STATUS_CHARGE) OR (Brusa2_Rx.StateAct = NLG_STATUS_CHARGE)) THEN
		chargeStatus := CHARGING;
		
	END_IF
	
// Charge plug not detected	
ELSE
	chargeStatus := NOT_CONNECTED;

END_IF

ACTION FreeContactor:
(*==============================================================================================================*)
(*    Uncomment this action to pulse the contactor free                                                         *)
(*==============================================================================================================*)
Pulsing := TRUE;                                               // Flag to stop Contactor control from running (main())

PulseTmr := PulseTmr + 1;                                      // Increment pulse timer every scan

IF (PulseTmr = PulseLength) THEN                               // Pulse length is number of 10ms scans
DO_q_Battery1ChargeMain_DO := NOT DO_q_Battery1ChargeMain_DO;  // Switch output
PulseTmr := 0;                                                 // Reset timer
END_IF
END_ACTION

END_PROGRAM

// Application/UserCode/BMS/OrionBMS/OrionBMS2_RxConversion
PROGRAM OrionBMS2_RxConversion
VAR
	Safety_OK   : BOOL;
END_VAR
VAR CONSTANT
	SYSTEMRX_CF	:	REAL	:=	0.1;
	CURRENT_CF	:	REAL	:=	0.1;
END_VAR

(*Convert input variables into real units by applying conversion factors and offsets*)

gr_OrionBMS2_PackVoltage			:=	UINT_TO_REAL(gu16_OrionBMS2_PackVoltage) * SYSTEMRX_CF;
gr_OrionBMS2_PackCurrent			:=	INT_TO_REAL(gs16_OrionBMS2_PackCurrent) * CURRENT_CF;
gr_OrionBMS2_PackSOC				:=	REAL_TO_USINT(gu8_OrionBMS2_RAW_SOC / 2);
gr_OrionBMS2_Max_Charging_Voltage	:= gu8_OrionBMS2_PopulatedCells *3.65;
	
OrionBMS2_DTCFlag1_0A07_DischargeLimitEnforcementFault1		:=	gu16_OrionBMS2_DTC_Flags1.0;
OrionBMS2_DTCFlag1_0A08_ChargerSafetyRelayFault1 			:=	gu16_OrionBMS2_DTC_Flags1.1;
OrionBMS2_DTCFlag1_0A09_InternalHardwareFault1				:=	gu16_OrionBMS2_DTC_Flags1.2;
OrionBMS2_DTCFlag1_0A0A_InternalHeatskinkThermistorFault 	:=	gu16_OrionBMS2_DTC_Flags1.3;
OrionBMS2_DTCFlag1_0A0B_InternalSoftwareFault1				:=	gu16_OrionBMS2_DTC_Flags1.4;
OrionBMS2_DTCFlag1_0A0C_HighestCellVoltageTooHighFault1 	:=	gu16_OrionBMS2_DTC_Flags1.5;
OrionBMS2_DTCFlag1_0A0E_LowestCellVoltageTooLowFault 		:=	gu16_OrionBMS2_DTC_Flags1.6;
OrionBMS2_DTCFlag1_0A10_PackTooHotFault1 					:=	gu16_OrionBMS2_DTC_Flags1.7;
OrionBMS2_DTCFlags_Reserved_Bit8 							:=	gu16_OrionBMS2_DTC_Flags1.8;
OrionBMS2_DTCFlags_Reserved_Bit9 							:=	gu16_OrionBMS2_DTC_Flags1.9;
OrionBMS2_DTCFlags_Reserved_Bit10 							:=	gu16_OrionBMS2_DTC_Flags1.10;
OrionBMS2_DTCFlags_Reserved_Bit11 							:=	gu16_OrionBMS2_DTC_Flags1.11;
OrionBMS2_DTCFlags_Reserved_Bit12 							:=	gu16_OrionBMS2_DTC_Flags1.12;
OrionBMS2_DTCFlags_Reserved_Bit13 							:=	gu16_OrionBMS2_DTC_Flags1.13;
OrionBMS2_DTCFlags_Reserved_Bit14 							:=	gu16_OrionBMS2_DTC_Flags1.14;
OrionBMS2_DTCFlags_Reserved_Bit15							:=	gu16_OrionBMS2_DTC_Flags1.15;

OrionBMS2_DTCFlags2_0A1F_InternalCommunicationFault			:=	gu16_OrionBMS2_DTC_Flags2.8;
OrionBMS2_DTCFlags2_0A12_CellBalancingStruckOffFault		:=	gu16_OrionBMS2_DTC_Flags2.9;
OrionBMS2_DTCFlags2_0A80_WeakCellFault						:=	gu16_OrionBMS2_DTC_Flags2.10;
OrionBMS2_DTCFlags2_0AFA_LowCellVoltageFault				:=	gu16_OrionBMS2_DTC_Flags2.11;
OrionBMS2_DTCFlags2_0A04_OpenWiringFault					:=	gu16_OrionBMS2_DTC_Flags2.12;
OrionBMS2_DTCFlags2_0AC0_CurrentSensorFault					:=	gu16_OrionBMS2_DTC_Flags2.13;
OrionBMS2_DTCFlags2_0A0D_HighestCellVoltageOver5vFault		:=	gu16_OrionBMS2_DTC_Flags2.14;
OrionBMS2_DTCFlags2_0A0F_CellASICFault						:=	gu16_OrionBMS2_DTC_Flags2.15;
OrionBMS2_DTCFlags2_0A02_WeakPackFault						:=	gu16_OrionBMS2_DTC_Flags2.0;
OrionBMS2_DTCFlags2_0A81_FanMonitorFault					:=	gu16_OrionBMS2_DTC_Flags2.1;
OrionBMS2_DTCFlags2_0A9C_ThermistorFault					:=	gu16_OrionBMS2_DTC_Flags2.2;
OrionBMS2_DTCFlags2_0100_ExternalCommunicationFault			:=	gu16_OrionBMS2_DTC_Flags2.3;
OrionBMS2_DTCFlags2_0560_RedundantPowerSupplyFault			:=	gu16_OrionBMS2_DTC_Flags2.4;
OrionBMS2_DTCFlags2_0AA6_HighVoltageIsolatonFault			:=	gu16_OrionBMS2_DTC_Flags2.5;
OrionBMS2_DTCFlags2_0A05_InputPowerSupplyFault				:=	gu16_OrionBMS2_DTC_Flags2.6;
OrionBMS2_DTCFlags2_0A06_ChargeLimitEnforcementFault		:=	gu16_OrionBMS2_DTC_Flags2.7;	
	
gq_BMS2_BalActive			:=	gu8_OrionBMS2_Custom_Flag_1.0;
gq_BMS2_Flag_1				:=	gu8_OrionBMS2_Custom_Flag_1.1;
gq_BMS2_Flag_2				:=	gu8_OrionBMS2_Custom_Flag_1.2;
gq_BMS2_Flag_3				:=	gu8_OrionBMS2_Custom_Flag_1.3;
gq_BMS2_Flag_4				:=	gu8_OrionBMS2_Custom_Flag_1.4;
gq_BMS2_Flag_5				:=	gu8_OrionBMS2_Custom_Flag_1.5;
gq_BMS2_Flag_6				:=	gu8_OrionBMS2_Custom_Flag_1.6;
Safety_OK    				:=	gu8_OrionBMS2_Custom_Flag_1.7;

END_PROGRAM

// Application/UserCode/CAN4/HMI_Rx
PROGRAM HMI_Rx
VAR
	HMI_Commands_Rx		      	:	Receive_CAN4_STD;
	gq_HMI_EStop_Bad			: BOOL;
	gq_Dennis_Handbrake     	: BOOL;
	StopChargeRq              	: BOOL;   // Stop charge request from HMI
	RAW_Pack_1_Balancing_Amps 	: BYTE;
	RAW_Pack_2_Balancing_Amps 	: BYTE;
	RAW_Pack_1_Offset_Volts	  	: BYTE;
	RAW_Pack_2_Offset_Volts   	: BYTE;
	Spare_6	                  	: BYTE;
	Spare_7                   	: BYTE;
	
END_VAR

(* From HMI *)
HMI_Commands_Rx(u32_COBID	:=	16#57B,
				q_NewData => ,
				au8_Data => ,
				u8_Length => 			);   (*8*)
				
gq_HMI_EStop_Bad			:=	HMI_Commands_Rx.au8_Data[0].0;
gq_Dennis_Handbrake			:=	HMI_Commands_Rx.au8_Data[0].1;
gq_HMI_Heater_Enable		:=	HMI_Commands_Rx.au8_Data[0].2;
StopChargeRq    			:=	HMI_Commands_Rx.au8_Data[0].3;
gq_HMI_Heater_Low			:=	HMI_Commands_Rx.au8_Data[0].4;
gq_HMI_Heater_Med			:=	HMI_Commands_Rx.au8_Data[0].5;
gq_HMI_Heater_Hi			:=	HMI_Commands_Rx.au8_Data[0].6;
qq_Spare_0_4				:=	HMI_Commands_Rx.au8_Data[0].7;

qq_BMS1_PB_DTC_Reset		:=	HMI_Commands_Rx.au8_Data[1].0;
qq_BMS2_PB_DTC_Reset		:=	HMI_Commands_Rx.au8_Data[1].1;
qq_Spare_1_2				:=	HMI_Commands_Rx.au8_Data[1].2;
qq_Spare_1_3				:=	HMI_Commands_Rx.au8_Data[1].3;
qq_Spare_1_4				:=	HMI_Commands_Rx.au8_Data[1].4;
qq_Spare_1_5				:=	HMI_Commands_Rx.au8_Data[1].5;
qq_Spare_1_6				:=	HMI_Commands_Rx.au8_Data[1].6;
qq_Spare_1_7				:=	HMI_Commands_Rx.au8_Data[1].7;
	
RAW_Pack_1_Balancing_Amps	:=	HMI_Commands_Rx.au8_Data[2]; 	// WIP
RAW_Pack_2_Balancing_Amps	:=	HMI_Commands_Rx.au8_Data[3];	// WIP
RAW_Pack_1_Offset_Volts		:=	HMI_Commands_Rx.au8_Data[4];	// WIP
RAW_Pack_2_Offset_Volts		:=	HMI_Commands_Rx.au8_Data[5];	// WIP
Spare_6						:=	HMI_Commands_Rx.au8_Data[6];
Spare_7						:=	HMI_Commands_Rx.au8_Data[7];

END_PROGRAM

// Application/UserCode/CAN Function Blocks/CAN4/Receive_CAN4_STD
FUNCTION_BLOCK Receive_CAN4_STD
VAR_INPUT
	u32_COBID	:	DWORD;
END_VAR
VAR_OUTPUT
	q_NewData	:	BOOL;
	au8_Data	:	ARRAY [0..7] OF BYTE;
	u8_Length	:	BYTE;
END_VAR
VAR
	hq_Initialise	:	BOOL	:=	FALSE;
	ht_RxMessage	:	t_CANReceive;
	ht_MsgRx		:	Callback_Receive_CAN1;
END_VAR



IF (hq_Initialise = FALSE) THEN
	(*
	IF (u32_COBID > 16#7FF) THEN
		(*29 bit*)
		;
	ELSE
		(*11 bit*)
		;
	END_IF
	*)
	
	(*11 bit*)
	G_CAN4_Channel.AddCOBID(i_CobId := u32_COBID,
							i_itfCallback := ht_MsgRx,
							i_Argument := ADR(ht_RxMessage));
	(*
	(*29 bit*)
	G_CAN4_Channel.AddCOBID(i_CobId := u32_COBID OR EPEC_CANVXD.MASK_29BIT,
							i_itfCallback := ht_MsgRx,
							i_Argument := ADR(ht_RxMessage));
*)	(*G_CAN4_Channel.SetMask(i_CobID := u32_COBID OR EPEC_CANVXD.MASK_29BIT, i_Mask := 16#0C009000 OR EPEC_CANVXD.MASK_29BIT);
*)
	hq_Initialise	:=	TRUE;
END_IF


IF (ht_RxMessage.q_NewDataRxed = TRUE) THEN
	au8_Data	:=	ht_RxMessage.Data;
	u8_Length	:=	ht_RxMessage.Len;
	q_NewData	:=	TRUE;
	ht_RxMessage.q_NewDataRxed	:=	FALSE;
ELSE
	q_NewData	:=	FALSE;
END_IF

END_FUNCTION_BLOCK

// Application/UserCode/Brusa/Brusa2_Comms/Brusa2_Rx
PROGRAM Brusa2_Rx
VAR
	ActAC_Rx	:	Receive_CAN3_STD;
	NLG2_ActErr_Rx	:	Receive_CAN3_STD;
	NLG2_ActInt_Rx	:	Receive_CAN3_STD;
	NLG2_ActLim_Rx	:	Receive_CAN3_STD;
	NLG2_ActPlug_Rx	:	Receive_CAN3_STD;
	
	ActAC_Rx_Timer		:	TON;
	ActErr_Rx_Timer		:	TON;
	ActInt_Rx_Timer		:	TON;
	ActLim_Rx_Timer		:	TON;
	ActPlug_Rx_Timer	:	TON;
	
	StatusPP_Rx			:	USINT; 
	StatusPP_Prev		:	USINT;
	
	ACVoltL1Act_Rx		:	USINT;
	ACVoltL2Act_Rx		:	USINT;
	ACVoltL3Act_Rx		:	USINT;
	ACFreqAct			:	USINT;
	SACPhaseRot			:	BOOL;
	ACCurrL1Act_Rx		:	USINT;
	ACCurrL2Act_Rx		:	USINT;
	ACCurrL3Act_Rx		:	USINT;
	ACPowTotAct_Rx		:	USINT;
	
	(*Act Err*)
	E_WrongHW					: BOOL;
	E_WrongFPGA					: BOOL;
	E_EPGAInit					: BOOL;
	E_NVSRam					: BOOL;
	E_Flash						: BOOL;
	E_OSTrap					: BOOL;
	E_HVIsoPos			: BOOL;
	E_HVIsoNeg			: BOOL;
	E_Internal			: BOOL;
	E_TempInt			: BOOL;
	E_DCHVVoltRed		: BOOL;
	E_IntSupply			: BOOL;
	E_CANMsgLost		: BOOL;
	E_CANValue			: BOOL;
	E_ACInterruption	: BOOL;
	E_DCHVVoltRange		: BOOL;
	E_TempCon			: BOOL;
	E_ConLocked			: BOOL;
	E_Interlock			: BOOL;
	E_Crash				: BOOL;
	E_PRELOAD			: BOOL;
	E_BURST				: BOOL;
	E_TPON				: BOOL;
	E_UZK				: BOOL;
	E_LatchFPGA					: BOOL;
	E_OverTemp					: BOOL;
	(*Warnings*)
	W_Watchdog					: BOOL;
	W_PowRed			: BOOL;
	W_TempInt			: BOOL;
	W_CANTimeout		: BOOL;
	W_CANOff			: BOOL;
	W_CANRx				: BOOL;
	W_CANTx				: BOOL;
	W_ConLocked			: BOOL;
	W_FPGA				: BOOL;
	W_ACVoltage			: BOOL;
	W_ACFrequency		: BOOL;
	W_PRELOAD			: BOOL;
	
	(*Act Int*)
	ACWhAct			:	UINT;
	DCHVWhAct			:	UINT;
	MaxTempAct_Rx		:	USINT;
	TempCon_Rx					:	USINT;
	DCHVAhAct_Rx				:	UINT;
	(*Act Lim*)
	StateCrtlPilot				:	USINT;
	DCHVVoltAct_Rx				:	UINT;
	StateAct					:	USINT; //0:Sleep 1:Wakeup 2:Standby 3:Ready2Charge 4:Charge 5:Shutdown
	S_DCHVCurrLim				:	BOOL;
	S_DCHVVoltLim				:	BOOL;
	DCHVCurrAct_Rx	:	UINT;
	S_ProximityLim		:	BOOL;
	S_CtrlPilotLim		:	BOOL;
	S_ConTempLim		:	BOOL;
	S_IntTempLim		:	BOOL;
	S_ACCurrLim			:	BOOL;
	ACCurrMaxAct_Rx		:	UINT;
	ACCurrHWAvl_Rx		:	USINT;
	S_ProximityDet		:	BOOL;
	S_CtrlPilotDet		:	BOOL;
	S_ConLocked			:	BOOL;
	S_ACDet				:	BOOL;
	S_HWWakeup			:	BOOL;
	S_HWEnablErre		:	BOOL;
	S_Err				:	BOOL;
	S_Warn				:	BOOL;
	(*Act Plug*)
	StatusCP			:	USINT;
	S_CPX1					:	BOOL;
	S_CPSCC				:	BOOL;
	ACCurrMaxCP_Rx	:	UINT;
	StatusPP			:	USINT; //0:PROXD_DETECTED 1:PROXD_CIRCUIT_RANGE 2:PROXD_CIRCUIT_LOW 3:PROXD_CIRCUIT_HIGH 4:PROXD_CIRCUIT_ERRATIC 5:PROXD_NOT_CONNECTED 7:SNA
	ACCurrMaxPP			:	USINT; //0:0 A 1:13 A 2:20 A 3:32 A 4:63 A 7:SNA
	s_ACVoltDerate		:	BOOL;
	S_ACDerating		:	BOOL;
	ACPhaseUsd			:	USINT;
	ACPhaseDet			:	USINT;  ///kak Why not used?????????
	CoolingRequest		:	USINT;
	TempCoolPlate_Rx	:	USINT; //Actual temperatur cool plate 255:SNA
	CommsLoss					:	BOOL;
	C_EnPhaseShift				:	BOOL;
END_VAR



ActAC_Rx(u32_COBID	:=	16#729,
				q_NewData => ,
				au8_Data => ,
				u8_Length => 			);
				
NLG2_ActErr_Rx(u32_COBID	:=	16#799,
				q_NewData => ,
				au8_Data => ,
				u8_Length => 			);
				
NLG2_ActInt_Rx(u32_COBID	:=	16#709,
				q_NewData => ,
				au8_Data => ,
				u8_Length => 			);
				
NLG2_ActLim_Rx(u32_COBID	:=	16#728,
				q_NewData => ,
				au8_Data => ,
				u8_Length => 			);
				
NLG2_ActPlug_Rx(u32_COBID	:=	16#739,
				q_NewData => ,
				au8_Data => ,
				u8_Length => 			);

(*Act AC*)
ACVoltL1Act_Rx		:=	ActAC_Rx.au8_Data[0];
ACVoltL2Act_Rx		:=	ActAC_Rx.au8_Data[1];
ACVoltL3Act_Rx		:=	ActAC_Rx.au8_Data[2];
ACFreqAct			:=	(ActAC_Rx.au8_Data[3] AND 2#01111111); (*Mask*)
SACPhaseRot			:=	ActAC_Rx.au8_Data[3].7;
ACCurrL1Act_Rx		:=	ActAC_Rx.au8_Data[4];
ACCurrL2Act_Rx		:=	ActAC_Rx.au8_Data[5];
ACCurrL3Act_Rx		:=	ActAC_Rx.au8_Data[6];
ACPowTotAct_Rx		:=	ActAC_Rx.au8_Data[7];;

(*Act Err*)
E_WrongHW			:=	NLG2_ActErr_Rx.au8_Data[0].0;
E_WrongFPGA			:=	NLG2_ActErr_Rx.au8_Data[0].1;
E_EPGAInit			:=	NLG2_ActErr_Rx.au8_Data[0].2;
E_NVSRam			:=	NLG2_ActErr_Rx.au8_Data[0].5;
E_Flash				:=	NLG2_ActErr_Rx.au8_Data[0].6;
E_OSTrap			:=	NLG2_ActErr_Rx.au8_Data[0].7;
E_HVIsoPos			:=	NLG2_ActErr_Rx.au8_Data[1].1;
E_HVIsoNeg			:=	NLG2_ActErr_Rx.au8_Data[1].2;
E_Internal			:=	NLG2_ActErr_Rx.au8_Data[1].4;
E_TempInt			:=	NLG2_ActErr_Rx.au8_Data[1].5;
E_DCHVVoltRed		:=	NLG2_ActErr_Rx.au8_Data[1].6;
E_IntSupply			:=	NLG2_ActErr_Rx.au8_Data[1].7;
E_CANMsgLost		:=	NLG2_ActErr_Rx.au8_Data[2].0;
E_CANValue			:=	NLG2_ActErr_Rx.au8_Data[2].1;
E_ACInterruption	:=	NLG2_ActErr_Rx.au8_Data[2].2;
E_DCHVVoltRange		:=	NLG2_ActErr_Rx.au8_Data[2].3;
E_TempCon			:=	NLG2_ActErr_Rx.au8_Data[2].4;
E_ConLocked			:=	NLG2_ActErr_Rx.au8_Data[2].5;
E_Interlock			:=	NLG2_ActErr_Rx.au8_Data[2].6;
E_Crash				:=	NLG2_ActErr_Rx.au8_Data[2].7;
E_PRELOAD			:=	NLG2_ActErr_Rx.au8_Data[3].1;
E_BURST				:=	NLG2_ActErr_Rx.au8_Data[3].2;
E_TPON				:=	NLG2_ActErr_Rx.au8_Data[3].3;
E_UZK				:=	NLG2_ActErr_Rx.au8_Data[3].4;
E_LatchFPGA			:=	NLG2_ActErr_Rx.au8_Data[3].5;
E_OverTemp			:=	NLG2_ActErr_Rx.au8_Data[3].7;
W_Watchdog			:=	NLG2_ActErr_Rx.au8_Data[4].7;
W_PowRed			:=	NLG2_ActErr_Rx.au8_Data[5].0;
W_TempInt			:=	NLG2_ActErr_Rx.au8_Data[5].1;
W_CANTimeout		:=	NLG2_ActErr_Rx.au8_Data[6].0;
W_CANOff			:=	NLG2_ActErr_Rx.au8_Data[6].1;
W_CANRx				:=	NLG2_ActErr_Rx.au8_Data[6].2;
W_CANTx				:=	NLG2_ActErr_Rx.au8_Data[6].3;
W_ConLocked			:=	NLG2_ActErr_Rx.au8_Data[6].7;
W_FPGA				:=	NLG2_ActErr_Rx.au8_Data[7].0;
W_ACVoltage			:=	NLG2_ActErr_Rx.au8_Data[7].1;
W_ACFrequency		:=	NLG2_ActErr_Rx.au8_Data[7].2;
W_PRELOAD			:=	NLG2_ActErr_Rx.au8_Data[7].3;


(*Act Int*)
ACWhAct			:=	SHL(USINT_TO_UINT(NLG2_ActInt_Rx.au8_Data[0]), 8) +
								USINT_TO_UINT(NLG2_ActInt_Rx.au8_Data[1]);
DCHVWhAct			:=	SHL(USINT_TO_UINT(NLG2_ActInt_Rx.au8_Data[2]), 8) +
								USINT_TO_UINT(NLG2_ActInt_Rx.au8_Data[3]);
MaxTempAct_Rx		:=	NLG2_ActInt_Rx.au8_Data[4];
TempCon_Rx			:=	NLG2_ActInt_Rx.au8_Data[5];
DCHVAhAct_Rx		:=	SHL(USINT_TO_UINT(NLG2_ActInt_Rx.au8_Data[6]), 8) +
								USINT_TO_UINT(NLG2_ActInt_Rx.au8_Data[7]);
(*Act Lim*)
StateCrtlPilot		:=	SHR((NLG2_ActLim_Rx.au8_Data[0] AND 2#11100000), 5);
DCHVVoltAct_Rx	:=	SHL(USINT_TO_UINT(NLG2_ActLim_Rx.au8_Data[0] AND 2#00011111), 8) +
								USINT_TO_UINT(NLG2_ActLim_Rx.au8_Data[1]);
StateAct			:=	SHR((NLG2_ActLim_Rx.au8_Data[2] AND 2#11100000), 5);
S_DCHVCurrLim		:=	NLG2_ActLim_Rx.au8_Data[2].4;
S_DCHVVoltLim		:=	NLG2_ActLim_Rx.au8_Data[2].3;
DCHVCurrAct_Rx	:=	SHL(USINT_TO_UINT(NLG2_ActLim_Rx.au8_Data[2] AND 2#00000111), 8) +
								USINT_TO_UINT(NLG2_ActLim_Rx.au8_Data[3]);
S_ProximityLim		:=	NLG2_ActLim_Rx.au8_Data[4].7;
S_CtrlPilotLim		:=	NLG2_ActLim_Rx.au8_Data[4].6;
S_ConTempLim		:=	NLG2_ActLim_Rx.au8_Data[4].5;
S_IntTempLim		:=	NLG2_ActLim_Rx.au8_Data[4].4;
S_ACCurrLim			:=	NLG2_ActLim_Rx.au8_Data[4].3;
ACCurrMaxAct_Rx	:=	SHL(USINT_TO_UINT(NLG2_ActLim_Rx.au8_Data[4] AND 2#00000111), 8) +
								USINT_TO_UINT(NLG2_ActLim_Rx.au8_Data[5]);
ACCurrHWAvl_Rx		:=	NLG2_ActLim_Rx.au8_Data[6];
S_ProximityDet		:=	NLG2_ActLim_Rx.au8_Data[7].7;
S_CtrlPilotDet		:=	NLG2_ActLim_Rx.au8_Data[7].6;
S_ConLocked			:=	NLG2_ActLim_Rx.au8_Data[7].5;
S_ACDet				:=	NLG2_ActLim_Rx.au8_Data[7].4;
S_HWWakeup			:=	NLG2_ActLim_Rx.au8_Data[7].3;
S_HWEnablErre		:=	NLG2_ActLim_Rx.au8_Data[7].2;
S_Err				:=	NLG2_ActLim_Rx.au8_Data[7].1;
S_Warn				:=	NLG2_ActLim_Rx.au8_Data[7].0;
(*Act Plug*)
StatusCP			:=	SHR((NLG2_ActPlug_Rx.au8_Data[0] AND 2#11100000), 5);
S_CPX1				:=	NLG2_ActPlug_Rx.au8_Data[0].4;
S_CPSCC				:=	NLG2_ActPlug_Rx.au8_Data[0].3;
ACCurrMaxCP_Rx	:=	SHL(USINT_TO_UINT(NLG2_ActPlug_Rx.au8_Data[0] AND 2#00000011), 8) +
								USINT_TO_UINT(NLG2_ActPlug_Rx.au8_Data[1]);
StatusPP			:=	SHR((NLG2_ActPlug_Rx.au8_Data[2] AND 2#01110000), 4);
ACCurrMaxPP		:=	NLG2_ActPlug_Rx.au8_Data[2] AND 2#00001111;
s_ACVoltDerate		:=	NLG2_ActPlug_Rx.au8_Data[4].7;
S_ACDerating		:=	NLG2_ActPlug_Rx.au8_Data[4].6;
ACPhaseUsd			:=	SHR((NLG2_ActPlug_Rx.au8_Data[4] AND 2#00111000), 3);
ACPhaseDet			:=	NLG2_ActPlug_Rx.au8_Data[4] AND 2#00000111;
CoolingRequest		:=	NLG2_ActPlug_Rx.au8_Data[5] AND 2#01111111;
TempCoolPlate_Rx	:=	NLG2_ActPlug_Rx.au8_Data[6];


IF (NOT(Brusa2_Tx.hton_NoPP_StopTx_Timer.Q) = TRUE) THEN
	ActAC_Rx_Timer(IN := NOT(ActAC_Rx.q_NewData), PT := T#5S);
	ActErr_Rx_Timer(IN := NOT(NLG2_ActErr_Rx.q_NewData), PT := T#5S);
	ActInt_Rx_Timer(IN := NOT(NLG2_ActInt_Rx.q_NewData), PT := T#5S);
	ActLim_Rx_Timer(IN := NOT(NLG2_ActLim_Rx.q_NewData), PT := T#5S);
	ActPlug_Rx_Timer(IN := NOT(NLG2_ActPlug_Rx.q_NewData), PT := T#5S);
	IF (ActAC_Rx_Timer.Q = TRUE AND ActErr_Rx_Timer.Q = TRUE AND ActInt_Rx_Timer.Q = TRUE AND
		ActLim_Rx_Timer.Q = TRUE AND ActPlug_Rx_Timer.Q = TRUE									) THEN
		CommsLoss	:=	TRUE;
	ELSE
		CommsLoss	:=	FALSE;
	END_IF
END_IF

Brusa1_RxConversion();

END_PROGRAM

// Application/UserCode/Brusa/Brusa2_Comms/Brusa2_Tx
PROGRAM Brusa2_Tx

VAR
	DenLim_Tx				:	EPEC_CANVXD.Msg;
	hu8_DenLim_Tx0			:	BYTE;
	hu8_DenLim_Tx2			:	BYTE;
	hu8_DenLim_Tx4			:	BYTE;
	hu8_DenLim_Tx6			:	BYTE;
	hton_Transmit_Timer		:	TON;
	hton_NoPP_StopTx_Timer	:	TON;
	StopBroadcast			:	BOOL;
	C_VentilRq				: 	BOOL;
END_VAR


Brusa2_TxConversion();

StopBroadcast	:=	(NOT(Brusa1_Rx.S_ProximityDet)(* AND DI_q_VehicleKL15_DI = FALSE*));
hton_NoPP_StopTx_Timer(IN := StopBroadcast, PT := T#1S);

// Brusa2_Control.C_Clr_Err	:= FALSE;
hu8_DenLim_Tx0	:=	UINT_TO_USINT(SHR(Brusa2_TxConversion.DCHVVoltLimMax_Tx, 8)) + SHL(BOOL_TO_USINT(C_VentilRq), 5) +
					SHL(BOOL_TO_USINT(Brusa.S_Unlock), 6) + SHL(BOOL_TO_USINT(Brusa.S_ErrClr), 7);
hu8_DenLim_Tx2	:=	(UINT_TO_USINT(SHR(Brusa2_TxConversion.DCHVCurrLimMax_Tx, 8)) AND 2#00000111) + SHL(Brusa.S_StateDem, 5);
hu8_DenLim_Tx4	:=	(UINT_TO_USINT(SHR(Brusa2_TxConversion.ACCurrLimMax_Tx, 8)) AND 2#00000111) + SHL(Brusa.LEDDem, 4);
//hu8_DenLim_Tx6	:=	(UINT_TO_USINT(SHR(Brusa2_TxConversion.ACPhaseShift_Tx, 8)) AND 2#00001111) + SHL(BOOL_TO_USINT(Brusa2_Rx.C_EnPhaseShift), 4);

DenLim_Tx.ID		:=	16#711;
DenLim_Tx.Data[0]	:=	hu8_DenLim_Tx0;
DenLim_Tx.Data[1]	:=	UINT_TO_USINT(Brusa2_TxConversion.DCHVVoltLimMax_Tx);
DenLim_Tx.Data[2]	:=	hu8_DenLim_Tx2;
DenLim_Tx.Data[3]	:=	UINT_TO_USINT(Brusa2_TxConversion.DCHVCurrLimMax_Tx);
DenLim_Tx.Data[4]	:=	hu8_DenLim_Tx4;
DenLim_Tx.Data[5]	:=	UINT_TO_USINT(Brusa2_TxConversion.ACCurrLimMax_Tx);
DenLim_Tx.Data[6]	:=	hu8_DenLim_Tx6;
DenLim_Tx.Data[7]	:=	UINT_TO_USINT(Brusa2_TxConversion.ACPhaseShift_Tx);
DenLim_Tx.Len		:=	8;



hton_Transmit_Timer(IN := NOT(hton_Transmit_Timer.Q), PT := T#90MS);
IF (hton_Transmit_Timer.Q = TRUE AND NOT(hton_NoPP_StopTx_Timer.Q) = TRUE) THEN
	G_CAN3_Channel.SendMessage(i_pMSG:=ADR(DenLim_Tx));
END_IF

END_PROGRAM

// Application/UserCode/Brusa/Brusa2_Comms/Brusa2_TxConversion
PROGRAM Brusa2_TxConversion
VAR
		DCHVVoltLimMax_Tx	:	UINT;
		DCHVCurrLimMax_Tx	:	UINT;
		ACCurrLimMax_Tx		:	UINT;
		ACPhaseShift_Tx		:	UINT;
END_VAR

//r2
DCHVVoltLimMax_Tx	:=	REAL_TO_UINT(Brusa.S_DCHVVoltLimMax / 0.1);
DCHVCurrLimMax_Tx	:=	REAL_TO_UINT((Brusa.S_DCHVCurrLimMax - 102.4) / 0.1);
ACCurrLimMax_Tx		:=	REAL_TO_UINT((Brusa.S_ACCurrLimMax - 102.4) / 0.1);
//ACPhaseShift_Tx		:=	REAL_TO_UINT(Brusa2_Control.ACPhaseShift / 0.1);

END_PROGRAM

// Application/UserCode/Brusa/Brusa1_Comms/Brusa1_RxConversion
PROGRAM Brusa1_RxConversion
VAR
	ACVoltL1Act		:	UINT;
	ACVoltL2Act		:	UINT;
	ACVoltL3Act		:	UINT;
	ACCurrL1Act		:	SINT;
	ACCurrL2Act		:	SINT;
	ACCurrL3Act		:	SINT;
	ACPowTotAct		:	UINT;
	MaxTempAct		:	INT;
	TempCon			:	INT;
	DCHVAhAct		:	REAL;
	DCHVVoltAct		:	REAL;
	DCHVCurrAct		:	REAL;
	ACCurrMaxAct	:	REAL;
	ACCurrHWAvl		:	REAL;
	ACCurrMaxCP		:	REAL;
	TempCoolPlate	:	INT;	
END_VAR

ACVoltL1Act	:=	USINT_TO_UINT(Brusa1_Rx.ACVoltL1Act_Rx) * 2;
ACVoltL2Act	:=	USINT_TO_UINT(Brusa1_Rx.ACVoltL2Act_Rx) * 2;
ACVoltL3Act	:=	USINT_TO_UINT(Brusa1_Rx.ACVoltL3Act_Rx) * 2;
ACCurrL1Act	:=	USINT_TO_SINT(Brusa1_Rx.ACCurrL1Act_Rx) - 127;
ACCurrL2Act	:=	USINT_TO_SINT(Brusa1_Rx.ACCurrL2Act_Rx) - 127;
ACCurrL3Act	:=	USINT_TO_SINT(Brusa1_Rx.ACCurrL3Act_Rx) - 127;
ACPowTotAct	:=	USINT_TO_UINT(Brusa1_Rx.ACPowTotAct_Rx) * 100;
MaxTempAct	:=	USINT_TO_INT(Brusa1_Rx.MaxTempAct_Rx) - 50;
TempCon		:=	USINT_TO_INT(Brusa1_Rx.TempCon_Rx) - 50;
DCHVAhAct		:=	UINT_TO_REAL(Brusa1_Rx.DCHVAhAct_Rx) * 0.01;
DCHVVoltAct		:=	UINT_TO_REAL(Brusa1_Rx.DCHVVoltAct_Rx) * 0.1;
DCHVCurrAct		:=	UINT_TO_REAL(Brusa1_Rx.DCHVCurrAct_Rx) * 0.1 - 100;
ACCurrMaxAct	:=	UINT_TO_REAL(Brusa1_Rx.ACCurrMaxAct_Rx) * 0.1 -100;
ACCurrHWAvl		:=	USINT_TO_REAL(Brusa1_Rx.ACCurrHWAvl_Rx) * 0.5;
ACCurrMaxCP		:=	UINT_TO_REAL(Brusa1_Rx.ACCurrMaxCP_Rx) * 0.1;
TempCoolPlate	:=	USINT_TO_INT(Brusa1_Rx.TempCoolPlate_Rx) - 50;

END_PROGRAM

// Application/UserCode/CAN Function Blocks/CAN3/Receive_CAN3_STD
FUNCTION_BLOCK Receive_CAN3_STD
VAR_INPUT
	u32_COBID	:	DWORD;
END_VAR
VAR_OUTPUT
	q_NewData	:	BOOL;
	au8_Data	:	ARRAY [0..7] OF BYTE;
	u8_Length	:	BYTE;
END_VAR
VAR
	hq_Initialise	:	BOOL	:=	FALSE;
	ht_RxMessage	:	t_CANReceive;
	ht_MsgRx		:	Callback_Receive_CAN1;
END_VAR



IF (hq_Initialise = FALSE) THEN
	(*
	IF (u32_COBID > 16#7FF) THEN
		(*29 bit*)
		;
	ELSE
		(*11 bit*)
		;
	END_IF
	*)
	
	(*11 bit*)
	G_CAN3_Channel.AddCOBID(i_CobId := u32_COBID,
							i_itfCallback := ht_MsgRx,
							i_Argument := ADR(ht_RxMessage));
	(*
	(*29 bit*)
	G_CAN3_Channel.AddCOBID(i_CobId := u32_COBID OR EPEC_CANVXD.MASK_29BIT,
							i_itfCallback := ht_MsgRx,
							i_Argument := ADR(ht_RxMessage));
*)	(*G_CAN3_Channel.SetMask(i_CobID := u32_COBID OR EPEC_CANVXD.MASK_29BIT, i_Mask := 16#0C009000 OR EPEC_CANVXD.MASK_29BIT);
*)
	hq_Initialise	:=	TRUE;
END_IF


IF (ht_RxMessage.q_NewDataRxed = TRUE) THEN
	au8_Data	:=	ht_RxMessage.Data;
	u8_Length	:=	ht_RxMessage.Len;
	q_NewData	:=	TRUE;
	ht_RxMessage.q_NewDataRxed	:=	FALSE;
ELSE
	q_NewData	:=	FALSE;
END_IF

END_FUNCTION_BLOCK

// Application/UserCode/BMS/BMSData
PROGRAM BMSData
VAR
	Batteries_Fully_Charged : BOOL;
	
	chargeInterlockFlt      : BOOL;
	
	firstPass               : R_TRIG;
END_VAR


IF (gu8_BMS_SOC >= 100 AND gs16_BMS2_CCL <= 0 AND gs16_BMS1_CCL <= 0) THEN
	Batteries_Fully_Charged				:=	TRUE;
ELSE
	Batteries_Fully_Charged				:=	FALSE;
END_IF

(*This program takes the slected BMS type and saves the relevent variables into the system values which are to be used*)
CASE gu8_BMSType OF
	BMS_ORION:
		gu8_BMS_SOC						:=	REAL_TO_USINT (MIN(gr_OrionBMS1_PackSOC, gr_OrionBMS2_PackSOC));
		gr_BMS_BatteryVoltage			:=	REAL_TO_UINT((gr_OrionBMS1_PackVoltage + gr_OrionBMS2_PackVoltage));
		gr_BMS1_Voltage					:=	REAL_TO_UINT(gr_OrionBMS1_PackVoltage);
		gr_BMS2_Voltage					:=	REAL_TO_UINT(gr_OrionBMS2_PackVoltage);
		gs16_BMS_BatteryCurrent			:=	REAL_TO_INT((gr_OrionBMS1_PackCurrent + gr_OrionBMS2_PackCurrent) / 2);
		gu16_BMS_Maximum_Pack_Voltage	:=	REAL_TO_UINT(gu16_OrionBMS1_MaximumPackVoltage + gu16_OrionBMS2_MaximumPackVoltage) / 10; (*Limit applied to prevent overcharging*)
		gs16_BMS1_CCL					:=	UINT_TO_INT(gu16_OrionBMS1_PackCCL);
		gs16_BMS2_CCL					:=	UINT_TO_INT(gu16_OrionBMS2_PackCCL);
		gu16_BMS_AverageCellVoltage		:=	(gu16_OrionBMS1_AverageCellVoltage + gu16_OrionBMS2_AverageCellVoltage) / 2;
		gu16_BMS_LowCellVoltage			:=	MIN(gu16_OrionBMS1_LowCellVoltage, gu16_OrionBMS2_LowCellVoltage);
		gu16_BMS_HighCellVoltage		:=	MAX(gu16_OrionBMS1_HighCellVoltage, gu16_OrionBMS2_HighCellVoltage);
		gr_BMS_AverageTemp				:=	(gu8_OrionBMS1_AverageTemp + gu8_OrionBMS2_AverageTemp) / 2;
		gr_BMS_LowTemp					:=	MIN(gu8_OrionBMS1_LowTemp, gu8_OrionBMS2_LowTemp);
		gr_BMS_HighTemp					:=	MAX(gu8_OrionBMS1_HighTemp, gu8_OrionBMS2_HighTemp);
		gr_BMS_DCL						:=	MIN(gu16_OrionBMS1_PackDCL, gu16_OrionBMS2_PackDCL);
		gr_BMS_CCL						:=	MIN(gu16_OrionBMS1_PackCCL, gu16_OrionBMS2_PackCCL);
		gu16_BMS_MinimumPackVoltage		:=	(gu16_OrionBMS1_MinimumPackVoltage + gu16_OrionBMS2_MinimumPackVoltage) / 10;
		gu16_BMS1_LowCellVoltage		:=	gu16_OrionBMS1_LowCellVoltage;
		gu16_BMS2_LowCellVoltage		:=	gu16_OrionBMS2_LowCellVoltage;
		gu16_BMS1_HighCellVoltage		:=	gu16_OrionBMS1_HighCellVoltage;
		gu16_BMS2_HighCellVoltage		:=	gu16_OrionBMS2_HighCellVoltage;
		gu16_BMS1_LowCellVoltage_ID		:=	gu8_OrionBMS1_LowCellVoltNumber;
		gu16_BMS2_LowCellVoltage_ID		:=	gu8_OrionBMS2_LowCellVoltNumber;
		gu16_BMS1_HighCellVoltage_ID	:=	gu8_OrionBMS1_HighCellVoltNumber;
		gu16_BMS2_HighCellVoltage_ID	:=	gu8_OrionBMS2_HighCellVoltNumber;
		
		
		
		
		
		
		
	
END_CASE

// Charge interlock fault used to stop drive mode selection when charge plug is inserted
// Resets on power cycle of VMU (first scan)
firstPass(CLK := TRUE);

IF firstPass.Q THEN
	chargeInterlockFlt := FALSE;
ELSIF gu16_OrionBMS1_FailsafeStatus.4 THEN
	chargeInterlockFlt := TRUE;
END_IF

END_PROGRAM

// Application/UserCode/Brusa/BrusaControl
(*===================================================================================================*)
(* Charger Control                                                                                   *)
(*===================================================================================================*)
FUNCTION_BLOCK BrusaControl
VAR_INPUT
(*Variable inputs ===================================================================================*)
	Master                  : BOOL;             // Master?
	Safety_OK               : BOOL;             // Battery safety ok signal
	CtrlPilotDet            : BOOL;
	ProximityDet            : BOOL;
	Error                   : BOOL;             // Brusa error
	ACDet                   : BOOL;
	BalancingActive         : BOOL; 
	StopChargeReq           : BOOL;             // Request to stop charging
	SysState                : BYTE;             // System state
	StateAct                : BYTE;             // Brusa recieved state
	Status                  : BYTE;             // Status PP?
	Balancing_Amps          : REAL;
	OffSet_Charge_Voltage   : REAL;
	CCL                     : REAL;
	MaxChargingVolts        : REAL;             // Max charging voltage from BMS
	ReportedMaxACCurr       : WORD;             // Reported AC max current from Brusa
	CPMaxAmps               : UINT;             // Control pilot allowable current
	
	
	
END_VAR
VAR_OUTPUT
	StateDem		        : USINT;           // Charger state request
	Unlock                  : BOOL;            // Charger unlock
	ErrorClearOut           : BOOL := FALSE;   // Request error clear
	StopCharging            : BOOL;            // Latch for stop charging request
	DCHVCurrLimMax			: REAL := 0;
	ACCurrLimMax			: REAL := 0;
	DCHVVoltLimMax			: REAL := 0;

END_VAR

VAR
	ChargerStates           :	tUpdate;         // Charger state machine variable
	
	ResetCnt                :   BYTE;            // Number of reset attempts

	ChargeDelayTmr          :   WORD;            // Scan counter to delay start charging 
	
	ResetOK     			:	BOOL;            // OK to reset
	
	CurrentLimit            :   REAL;            // Maximum allowable current
			
END_VAR

VAR CONSTANT

(*Charger control words ============================================================================*)
	NLG_CONTROL_STANDBY		:	USINT	:=	0;    // Standby request
	NLG_CONTROL_CHARGE		:	USINT	:=	1;	  // Charge request
	NLG_CONTROL_SLEEP		:	USINT	:=	6;    // Sleep request
	NLG_CONTROL_SNA			:	USINT	:=	7;    
	
(*Charger status words =============================================================================*)
	NLG_STATUS_SLEEP		:	USINT	:=	0;
	NLG_STATUS_WAKEUP		:	USINT	:=	1;
	NLG_STATUS_STANDBY		:	USINT	:=	2;
	NLG_STATUS_READY2CHARGE	:	USINT	:=	3;
	NLG_STATUS_CHARGE		:	USINT	:=	4;
	NLG_STATUS_SHUTDOWN		:	USINT	:=	5;
	
(* Case step constants =============================================================================*)
	_Sleep                  :   BYTE    := 0;
	_Standby                :   BYTE 	:= 1;
	_Charging               :   BYTE    := 2;
	_Error                  :   BYTE    := 255;
	
(* Charger plug in states ==========================================================================*)
	CHARGER_DETECTED		:	BYTE	:=	0;
	CHARGER_NOTCONNECTED	:	BYTE	:=	5;
	
	PP_32A					:	BYTE	:=	3;
	PP_64A					:	BYTE	:=	4;
	
END_VAR

(*===================================================================================================*)
(* Charger state machine                                                                             *)
(*===================================================================================================*)

// Discuss error clearing - looks like error clear message is always set to false

(* Handle charge lock request =======================================================================*)	
IF (StopChargeReq) THEN                        // Move to standy if charge stop requested from HMI
	StopCharging := TRUE;
ELSIF (StopCharging AND NOT ProximityDet) THEN // Only allow charging once the charge plug has been removed and reinserted
	StopCharging := FALSE;
END_IF

CASE ChargerStates.Step OF
(* Sleep state ======================================================================================*)	
_Sleep:
	
	Unlock := TRUE;                           // Unlock charge plug

	IF (StateAct <> 0) THEN                   // Moved out of sleep state into wakeup state
		ChargerStates.Next := _Standby;       // Move to standby state 
	END_IF
	
(* Standby state ====================================================================================*)	
_Standby:
		
	Unlock := TRUE;                                          // Unlock charge plug
		
	IF OkToCharge() THEN                                     // Charging conditions OK (If charging conditions are met then lock should engage automatically)
		Unlock := FALSE;                                     // Allow charger to lock
		IF (StateAct = NLG_STATUS_READY2CHARGE) OR (StateAct = NLG_STATUS_CHARGE) THEN
		ChargerStates.Next := _Charging;                     // Move to charging state
		END_IF
	ELSIF (Error) THEN
		ChargerStates.Next := _Error;                        // Move to error state
	ELSIF (StateAct = NLG_STATUS_SLEEP) THEN
		ChargerStates.Next := _Sleep;                        // Move to sleep state
	ELSE
		StateDem :=	NLG_CONTROL_STANDBY;                     // Set STANDBY state
	END_IF
	
(* Charging state ===================================================================================*)
_Charging:
	
	StateDem :=	NLG_CONTROL_CHARGE;          // Set CHARGING state 

	IF NOT (OkToCharge()) THEN               // If not ok to charge check for errors
		
		IF (Error) THEN
			ChargerStates.Next := _Error;    // Move to error state 
		ELSE
			ChargerStates.Next := _Standby;  // Move back to standby state 
		END_IF
		
	END_IF
	
(* Error state ======================================================================================*)
_Error:

		IF (OkToReset()) THEN	
			
			ErrorClearOut := SEL((ChargerStates.Tmr < 100), FALSE, TRUE); // Request error clear
			
			IF (ChargerStates.Tmr > 6000) THEN   // 1 min - charger requires 1 min to attempt automatic recovery or temp recovery
				ResetCnt   := ResetCnt +1;       // Increment reset count
				ChargerStates.Next := _Standby;  // Move back to Standby state	
			END_IF
			
		END_IF	
	
END_CASE

(*Set the DC current limit depending on balancing status ==========================================*)
DCHVCurrLimMax := SEL( BalancingActive, CCL, MIN(CCL, Balancing_Amps));

(*Set the AC current limit based on the wire that is plugged in ===================================*)
IF (Brusa1_Rx.ACCurrMaxPP = PP_32A) THEN
	CurrentLimit	:=	MIN(15, ((CPMaxAmps/20)-1));    // Div by 200 to get single side and A from mA, then -1 for lead acid battery
ELSIF (Brusa1_Rx.ACCurrMaxPP = PP_64A) THEN
	CurrentLimit	:=	MIN(28, ((CPMaxAmps/20)-1));    // Div by 200 to get single side and A from mA, then -1 for lead acid battery
ELSE
	CurrentLimit	:=	0;
END_IF

(* Delay charge and then ramp current up to max - Add 50mA each scan ==============================*)

// If available currrent limit drops then drop requested current immediately
IF (ACCurrLimMax > CurrentLimit) THEN
	ACCurrLimMax := CurrentLimit;
	
// If available current is less than requested increase by 50mA each scan (e.g. 30Amps achieved in 6s)
ELSIF (ACCurrLimMax < CurrentLimit) THEN
	ACCurrLimMax := ACCurrLimMax + 0.005;

// Otherwise request the maximum allowable current
ELSE
	ACCurrLimMax := CurrentLimit;
END_IF

(* Limit maximum voltage to be delivered to each pack =============================================*)
DCHVVoltLimMax	:=	(MaxChargingVolts); // - OffSet_Charge_Voltage); 

Update(ADR(ChargerStates));                                     // State machine update

(*===================================================================================================*)
(* Monitor charging conditions                                                                       *)
(*===================================================================================================*)
METHOD OkToCharge : BOOL
VAR_INPUT
END_VAR
(*===================================================================================================*)
(* Monitor charging conditions                                                                       *)
(*===================================================================================================*)
OkToCharge := ((Safety_OK                                                              AND  // Check BMS safety is OK
              (CtrlPilotDet OR ACDet)                                                  AND  // Check for Control pilot or ACHV
	          (ProximityDet                                                            AND  // Check plug proximity detect
			  (Status = CHARGER_DETECTED)                                              AND  // Check staus charger detected
			   NOT (Error OR StopChargeReq OR StopCharging))));                             // Check there are no errors or stop charge request
END_METHOD

